LIN {X 0,Y 245.794,Z 1176.659,A -85,B 0,C 180,E1 11030.463,E2 11030.463} C_VEL
LIN {X 0,Y 253.658,Z 1155.772,A -85,B 0,C 180,E1 11026.264,E2 11026.264} C_VEL
LIN {X 0,Y 262.655,Z 1132.428,A -85,B 0,C 180,E1 11022.399,E2 11022.399} C_VEL
LIN {X 0,Y 271.964,Z 1108.253,A -85,B 0,C 180,E1 11019.132,E2 11019.132} C_VEL
LIN {X 0,Y 282.858,Z 1079.724,A -85,B 0,C 180,E1 11015.958,E2 11015.958} C_VEL
LIN {X 0,Y 293.467,Z 1051.429,A -85,B 0,C 180,E1 11013.416,E2 11013.416} C_VEL
LIN {X 0,Y 303.782,Z 1022.552,A -85,B 0,C 180,E1 11011.336,E2 11011.336} C_VEL
LIN {X 0,Y 309.269,Z 1005.972,A -85,B 0,C 180,E1 11010.325,E2 11010.325} C_VEL
LIN {X 0,Y 306.49,Z 980.098,A -85,B 0,C 180,E1 11007.282,E2 11007.282} C_VEL
LIN {X 0,Y 305.142,Z 955.248,A -85,B 0,C 180,E1 11004.695,E2 11004.695} C_VEL
LIN {X 0,Y 304.735,Z 928.08,A -85,B 0,C 180,E1 11002.235,E2 11002.235} C_VEL
LIN {X 0,Y 305.285,Z 899.503,A -85,B 0,C 180,E1 11000.074,E2 11000.074} C_VEL
LIN {X 0,Y 306.681,Z 870.662,A -85,B 0,C 180,E1 10998.043,E2 10998.043} C_VEL
LIN {X 0,Y 314.524,Z 847.538,A -85,B 0,C 180,E1 10995.016,E2 10995.016} C_VEL
LIN {X 0,Y 309.833,Z 833.339,A -85,B 0,C 180,E1 10991.165,E2 10991.165} C_VEL
LIN {X 0,Y 304.885,Z 819.165,A -85,B 0,C 180,E1 10986.97,E2 10986.97} C_VEL
LIN {X 0,Y 300.201,Z 806.583,A -85,B 0,C 180,E1 10982.864,E2 10982.864} C_VEL
LIN {X 0,Y 295.689,Z 794.743,A -85,B 0,C 180,E1 10978.644,E2 10978.644} C_VEL
LIN {X 0,Y 291.025,Z 783.188,A -85,B 0,C 180,E1 10974.084,E2 10974.084} C_VEL
LIN {X 0,Y 286.711,Z 772.817,A -85,B 0,C 180,E1 10969.545,E2 10969.545} C_VEL
LIN {X 0,Y 282.704,Z 763.649,A -85,B 0,C 180,E1 10965.037,E2 10965.037} C_VEL
LIN {X 0,Y 279.359,Z 756.044,A -85,B 0,C 180,E1 10960.884,E2 10960.884} C_VEL
LIN {X 0,Y 276.382,Z 749.179,A -85,B 0,C 180,E1 10956.759,E2 10956.759} C_VEL
LIN {X 0,Y 274.386,Z 744.79,A -85,B 0,C 180,E1 10953.778,E2 10953.778} C_VEL
LIN {X 0,Y 281.502,Z 746.329,A -85,B 0,C 180,E1 10950.823,E2 10950.823} C_VEL
LIN {X 0,Y 285.736,Z 758.772,A -85,B 0,C 180,E1 10947.391,E2 10947.391} C_VEL
LIN {X 0,Y 289.434,Z 771.953,A -85,B 0,C 180,E1 10944.27,E2 10944.27} C_VEL
LIN {X 0,Y 291.796,Z 781.823,A -85,B 0,C 180,E1 10942.234,E2 10942.234} C_VEL
LIN {X 0,Y 283.399,Z 830.233,A -85,B 0,C 180,E1 10937.505,E2 10937.505} C_VEL
LIN {X 0,Y 275.294,Z 882,A -85,B 0,C 180,E1 10932.497,E2 10932.497} C_VEL
LIN {X 0,Y 275.45,Z 888.928,A -85,B 0,C 180,E1 10932.221,E2 10932.221} C_VEL
LIN {X 0,Y 266.995,Z 1035.963,A -85,B 0,C 180,E1 10928.695,E2 10928.695} C_VEL
LIN {X 0,Y 266,Z 1058.102,A -85,B 0,C 180,E1 10927.978,E2 10927.978} C_VEL
LIN {X 0,Y 264.246,Z 1076.059,A -85,B 0,C 180,E1 10927.021,E2 10927.021} C_VEL
LIN {X 0,Y 261.729,Z 1092.625,A -85,B 0,C 180,E1 10925.764,E2 10925.764} C_VEL
LIN {X 0,Y 258.407,Z 1108.653,A -85,B 0,C 180,E1 10924.126,E2 10924.126} C_VEL
LIN {X 0,Y 254.379,Z 1124.313,A -85,B 0,C 180,E1 10922.045,E2 10922.045} C_VEL
LIN {X 0,Y 250.173,Z 1138.097,A -85,B 0,C 180,E1 10919.705,E2 10919.705} C_VEL
LIN {X 0,Y 245.84,Z 1150.471,A -85,B 0,C 180,E1 10917.035,E2 10917.035} C_VEL
LIN {X 0,Y 241.448,Z 1161.815,A -85,B 0,C 180,E1 10913.94,E2 10913.94} C_VEL
LIN {X 0,Y 237.312,Z 1171.782,A -85,B 0,C 180,E1 10910.466,E2 10910.466} C_VEL
LIN {X 0,Y 233.669,Z 1180.12,A -85,B 0,C 180,E1 10906.657,E2 10906.657} C_VEL
LIN {X 0,Y 230.699,Z 1186.833,A -85,B 0,C 180,E1 10902.512,E2 10902.512} C_VEL
LIN {X 0,Y 228.64,Z 1191.633,A -85,B 0,C 180,E1 10898.294,E2 10898.294} C_VEL
LIN {X 0,Y 227.421,Z 1194.668,A -85,B 0,C 180,E1 10894.03,E2 10894.03} C_VEL
LIN {X 0,Y 226.961,Z 1196.042,A -85,B 0,C 180,E1 10889.492,E2 10889.492} C_VEL
LIN {X 0,Y 227.297,Z 1195.648,A -85,B 0,C 180,E1 10884.949,E2 10884.949} C_VEL
LIN {X 0,Y 228.487,Z 1193.456,A -85,B 0,C 180,E1 10880.424,E2 10880.424} C_VEL
LIN {X 0,Y 230.473,Z 1189.568,A -85,B 0,C 180,E1 10876.192,E2 10876.192} C_VEL
LIN {X 0,Y 233.392,Z 1183.816,A -85,B 0,C 180,E1 10872.006,E2 10872.006} C_VEL
LIN {X 0,Y 237.05,Z 1176.45,A -85,B 0,C 180,E1 10868.122,E2 10868.122} C_VEL
LIN {X 0,Y 241.081,Z 1167.875,A -85,B 0,C 180,E1 10864.707,E2 10864.707} C_VEL
LIN {X 0,Y 245.543,Z 1157.661,A -85,B 0,C 180,E1 10861.544,E2 10861.544} C_VEL
LIN {X 0,Y 250.186,Z 1145.999,A -85,B 0,C 180,E1 10858.694,E2 10858.694} C_VEL
LIN {X 0,Y 254.869,Z 1132.781,A -85,B 0,C 180,E1 10856.142,E2 10856.142} C_VEL
LIN {X 0,Y 259.222,Z 1118.358,A -85,B 0,C 180,E1 10853.965,E2 10853.965} C_VEL
LIN {X 0,Y 263.101,Z 1102.793,A -85,B 0,C 180,E1 10852.135,E2 10852.135} C_VEL
LIN {X 0,Y 266.253,Z 1086.649,A -85,B 0,C 180,E1 10850.68,E2 10850.68} C_VEL
LIN {X 0,Y 267.79,Z 1076.701,A -85,B 0,C 180,E1 10849.969,E2 10849.969} C_VEL
LIN {X 0,Y 270.006,Z 1077.25,A -85,B 0,C 180,E1 10849.601,E2 10849.601} C_VEL
LIN {X 0,Y 273.138,Z 1076.234,A -85,B 0,C 180,E1 10849.334,E2 10849.334} C_VEL
LIN {X 0,Y 277.103,Z 1073.311,A -85,B 0,C 180,E1 10849.22,E2 10849.22} C_VEL
LIN {X 0,Y 279.582,Z 1072.671,A -85,B 0,C 180,E1 10848.992,E2 10848.992} C_VEL
LIN {X 0,Y 272.711,Z 1094.804,A -85,B 0,C 180,E1 10846.636,E2 10846.636} C_VEL
LIN {X 0,Y 265.454,Z 1115.949,A -85,B 0,C 180,E1 10843.874,E2 10843.874} C_VEL
LIN {X 0,Y 257.942,Z 1136.201,A -85,B 0,C 180,E1 10840.635,E2 10840.635} C_VEL
LIN {X 0,Y 251.122,Z 1153.816,A -85,B 0,C 180,E1 10837.214,E2 10837.214} C_VEL
LIN {X 0,Y 244.423,Z 1170.711,A -85,B 0,C 180,E1 10833.242,E2 10833.242} C_VEL
LIN {X 0,Y 238.202,Z 1186.646,A -85,B 0,C 180,E1 10828.675,E2 10828.675} C_VEL
LIN {X 0,Y 233.894,Z 1198.218,A -85,B 0,C 180,E1 10824.67,E2 10824.67} C_VEL
LIN {X 0,Y 231.503,Z 1202.313,A -85,B 0,C 180,E1 10823.15,E2 10823.15} C_VEL
LIN {X 0,Y 222.063,Z 1212.153,A -85,B 0,C 180,E1 10819.027,E2 10819.027} C_VEL
LIN {X 0,Y 220.419,Z 1215.207,A -85,B 0,C 180,E1 10817.547,E2 10817.547} C_VEL
LIN {X 0,Y 218.075,Z 1224.725,A -85,B 0,C 180,E1 10812.176,E2 10812.176} C_VEL
LIN {X 0,Y 216.806,Z 1232.767,A -85,B 0,C 180,E1 10806.621,E2 10806.621} C_VEL
LIN {X 0,Y 216.41,Z 1238.955,A -85,B 0,C 180,E1 10801.324,E2 10801.324} C_VEL
LIN {X 0,Y 216.474,Z 1243.705,A -85,B 0,C 180,E1 10796.027,E2 10796.027} C_VEL
LIN {X 0,Y 217.079,Z 1247.526,A -85,B 0,C 180,E1 10790.455,E2 10790.455} C_VEL
LIN {X 0,Y 218.97,Z 1250.36,A -85,B 0,C 180,E1 10784.099,E2 10784.099} C_VEL
LIN {X 0,Y 223.396,Z 1251.95,A -85,B 0,C 180,E1 10777.083,E2 10777.083} C_VEL
LIN {X 0,Y 231.352,Z 1251.855,A -85,B 0,C 180,E1 10769.911,E2 10769.911} C_VEL
LIN {X 0,Y 243.153,Z 1249.952,A -85,B 0,C 180,E1 10763.103,E2 10763.103} C_VEL
LIN {X 0,Y 258.957,Z 1246.212,A -85,B 0,C 180,E1 10756.887,E2 10756.887} C_VEL
LIN {X 0,Y 264.381,Z 1244.756,A -85,B 0,C 180,E1 10755.163,E2 10755.163} C_VEL
LIN {X 0,Y 246.171,Z 1253.178,A -85,B 0,C 180,E1 10749.322,E2 10749.322} C_VEL
LIN {X 0,Y 232.274,Z 1260.245,A -85,B 0,C 180,E1 10742.558,E2 10742.558} C_VEL
LIN {X 0,Y 223.251,Z 1265.258,A -85,B 0,C 180,E1 10735.469,E2 10735.469} C_VEL
LIN {X 0,Y 218.472,Z 1268.085,A -85,B 0,C 180,E1 10728.668,E2 10728.668} C_VEL
LIN {X 0,Y 216.631,Z 1269.015,A -85,B 0,C 180,E1 10722.262,E2 10722.262} C_VEL
LIN {X 0,Y 216.607,Z 1268.218,A -85,B 0,C 180,E1 10716.364,E2 10716.364} C_VEL
LIN {X 0,Y 217.109,Z 1266.169,A -85,B 0,C 180,E1 10711.587,E2 10711.587} C_VEL
LIN {X 0,Y 217.301,Z 1263.421,A -85,B 0,C 180,E1 10707.63,E2 10707.63} C_VEL
LIN {X 0,Y 217.222,Z 1259.203,A -85,B 0,C 180,E1 10703.396,E2 10703.396} C_VEL
LIN {X 0,Y 217.27,Z 1252.953,A -85,B 0,C 180,E1 10698.59,E2 10698.59} C_VEL
LIN {X 0,Y 217.992,Z 1244.563,A -85,B 0,C 180,E1 10693.466,E2 10693.466} C_VEL
LIN {X 0,Y 219.847,Z 1233.738,A -85,B 0,C 180,E1 10688.107,E2 10688.107} C_VEL
LIN {X 0,Y 223.25,Z 1220.001,A -85,B 0,C 180,E1 10682.532,E2 10682.532} C_VEL
LIN {X 0,Y 227.725,Z 1205.387,A -85,B 0,C 180,E1 10677.615,E2 10677.615} C_VEL
LIN {X 0,Y 234.276,Z 1186.649,A -85,B 0,C 180,E1 10672.392,E2 10672.392} C_VEL
LIN {X 0,Y 242.106,Z 1165.933,A -85,B 0,C 180,E1 10667.669,E2 10667.669} C_VEL
LIN {X 0,Y 250.586,Z 1144.273,A -85,B 0,C 180,E1 10663.618,E2 10663.618} C_VEL
LIN {X 0,Y 259.832,Z 1120.935,A -85,B 0,C 180,E1 10660.028,E2 10660.028} C_VEL
LIN {X 0,Y 271.037,Z 1092.34,A -85,B 0,C 180,E1 10656.47,E2 10656.47} C_VEL
LIN {X 0,Y 282.4,Z 1063.011,A -85,B 0,C 180,E1 10653.528,E2 10653.528} C_VEL
LIN {X 0,Y 292.968,Z 1034.784,A -85,B 0,C 180,E1 10651.25,E2 10651.25} C_VEL
LIN {X 0,Y 302.537,Z 1007.602,A -85,B 0,C 180,E1 10649.502,E2 10649.502} C_VEL
LIN {X 0,Y 300.088,Z 981.059,A -85,B 0,C 180,E1 10646.305,E2 10646.305} C_VEL
LIN {X 0,Y 299.039,Z 955.864,A -85,B 0,C 180,E1 10643.637,E2 10643.637} C_VEL
LIN {X 0,Y 299.042,Z 928.661,A -85,B 0,C 180,E1 10641.121,E2 10641.121} C_VEL
LIN {X 0,Y 299.948,Z 898.691,A -85,B 0,C 180,E1 10638.829,E2 10638.829} C_VEL
LIN {X 0,Y 301.641,Z 868.509,A -85,B 0,C 180,E1 10636.679,E2 10636.679} C_VEL
LIN {X 0,Y 307.857,Z 850.994,A -85,B 0,C 180,E1 10634.387,E2 10634.387} C_VEL
LIN {X 0,Y 303,Z 836.151,A -85,B 0,C 180,E1 10630.265,E2 10630.265} C_VEL
LIN {X 0,Y 297.902,Z 821.422,A -85,B 0,C 180,E1 10625.779,E2 10625.779} C_VEL
LIN {X 0,Y 293.033,Z 808.289,A -85,B 0,C 180,E1 10621.363,E2 10621.363} C_VEL
LIN {X 0,Y 288.537,Z 796.595,A -85,B 0,C 180,E1 10617.02,E2 10617.02} C_VEL
LIN {X 0,Y 284.155,Z 785.659,A -85,B 0,C 180,E1 10612.519,E2 10612.519} C_VEL
LIN {X 0,Y 279.79,Z 775.02,A -85,B 0,C 180,E1 10607.618,E2 10607.618} C_VEL
LIN {X 0,Y 275.831,Z 765.954,A -85,B 0,C 180,E1 10602.925,E2 10602.925} C_VEL
LIN {X 0,Y 272.611,Z 758.595,A -85,B 0,C 180,E1 10598.68,E2 10598.68} C_VEL
LIN {X 0,Y 270.256,Z 753.347,A -85,B 0,C 180,E1 10595.287,E2 10595.287} C_VEL
LIN {X 0,Y 269.775,Z 751.899,A -85,B 0,C 180,E1 10594.301,E2 10594.301} C_VEL
LIN {X 0,Y 277.293,Z 753.26,A -85,B 0,C 180,E1 10591.106,E2 10591.106} C_VEL
LIN {X 0,Y 281.203,Z 765.326,A -85,B 0,C 180,E1 10587.767,E2 10587.767} C_VEL
LIN {X 0,Y 284.748,Z 778.734,A -85,B 0,C 180,E1 10584.592,E2 10584.592} C_VEL
LIN {X 0,Y 286.108,Z 785.803,A -85,B 0,C 180,E1 10583.154,E2 10583.154} C_VEL
LIN {X 0,Y 277.26,Z 835.51,A -85,B 0,C 180,E1 10578.284,E2 10578.284} C_VEL
LIN {X 0,Y 269.532,Z 883.178,A -85,B 0,C 180,E1 10573.64,E2 10573.64} C_VEL
LIN {X 0,Y 269.648,Z 889.812,A -85,B 0,C 180,E1 10573.372,E2 10573.372} C_VEL
LIN {X 0,Y 260.896,Z 1036.324,A -85,B 0,C 180,E1 10569.816,E2 10569.816} C_VEL
LIN {X 0,Y 259.821,Z 1059.023,A -85,B 0,C 180,E1 10569.071,E2 10569.071} C_VEL
LIN {X 0,Y 257.987,Z 1077.015,A -85,B 0,C 180,E1 10568.096,E2 10568.096} C_VEL
LIN {X 0,Y 255.337,Z 1093.738,A -85,B 0,C 180,E1 10566.804,E2 10566.804} C_VEL
LIN {X 0,Y 251.881,Z 1109.729,A -85,B 0,C 180,E1 10565.138,E2 10565.138} C_VEL
LIN {X 0,Y 247.896,Z 1124.657,A -85,B 0,C 180,E1 10563.126,E2 10563.126} C_VEL
LIN {X 0,Y 243.507,Z 1138.558,A -85,B 0,C 180,E1 10560.741,E2 10560.741} C_VEL
LIN {X 0,Y 238.88,Z 1151.282,A -85,B 0,C 180,E1 10557.952,E2 10557.952} C_VEL
LIN {X 0,Y 234.216,Z 1162.823,A -85,B 0,C 180,E1 10554.728,E2 10554.728} C_VEL
LIN {X 0,Y 229.89,Z 1172.782,A -85,B 0,C 180,E1 10551.158,E2 10551.158} C_VEL
LIN {X 0,Y 226.071,Z 1181.107,A -85,B 0,C 180,E1 10547.234,E2 10547.234} C_VEL
LIN {X 0,Y 222.952,Z 1187.812,A -85,B 0,C 180,E1 10542.954,E2 10542.954} C_VEL
LIN {X 0,Y 220.784,Z 1192.605,A -85,B 0,C 180,E1 10538.591,E2 10538.591} C_VEL
LIN {X 0,Y 219.5,Z 1195.629,A -85,B 0,C 180,E1 10534.176,E2 10534.176} C_VEL
LIN {X 0,Y 219.018,Z 1196.997,A -85,B 0,C 180,E1 10529.473,E2 10529.473} C_VEL
LIN {X 0,Y 219.38,Z 1196.596,A -85,B 0,C 180,E1 10524.766,E2 10524.766} C_VEL
LIN {X 0,Y 220.549,Z 1194.562,A -85,B 0,C 180,E1 10520.34,E2 10520.34} C_VEL
LIN {X 0,Y 222.602,Z 1190.789,A -85,B 0,C 180,E1 10515.959,E2 10515.959} C_VEL
LIN {X 0,Y 225.604,Z 1185.164,A -85,B 0,C 180,E1 10511.655,E2 10511.655} C_VEL
LIN {X 0,Y 229.328,Z 1178.024,A -85,B 0,C 180,E1 10507.705,E2 10507.705} C_VEL
LIN {X 0,Y 233.599,Z 1169.435,A -85,B 0,C 180,E1 10504.11,E2 10504.11} C_VEL
LIN {X 0,Y 238.433,Z 1158.873,A -85,B 0,C 180,E1 10500.724,E2 10500.724} C_VEL
LIN {X 0,Y 243.421,Z 1146.868,A -85,B 0,C 180,E1 10497.721,E2 10497.721} C_VEL
LIN {X 0,Y 248.299,Z 1133.631,A -85,B 0,C 180,E1 10495.119,E2 10495.119} C_VEL
LIN {X 0,Y 252.828,Z 1119.174,A -85,B 0,C 180,E1 10492.904,E2 10492.904} C_VEL
LIN {X 0,Y 256.861,Z 1103.573,A -85,B 0,C 180,E1 10491.044,E2 10491.044} C_VEL
LIN {X 0,Y 260.061,Z 1087.795,A -85,B 0,C 180,E1 10489.602,E2 10489.602} C_VEL
LIN {X 0,Y 260.438,Z 1086.527,A -85,B 0,C 180,E1 10489.463,E2 10489.463} C_VEL
LIN {X 0,Y 262.674,Z 1087.016,A -85,B 0,C 180,E1 10489.097,E2 10489.097} C_VEL
LIN {X 0,Y 265.828,Z 1086.116,A -85,B 0,C 180,E1 10488.831,E2 10488.831} C_VEL
LIN {X 0,Y 269.275,Z 1084.016,A -85,B 0,C 180,E1 10488.704,E2 10488.704} C_VEL
LIN {X 0,Y 262.103,Z 1105.434,A -85,B 0,C 180,E1 10486.139,E2 10486.139} C_VEL
LIN {X 0,Y 254.799,Z 1125.376,A -85,B 0,C 180,E1 10483.219,E2 10483.219} C_VEL
LIN {X 0,Y 247.46,Z 1144.296,A -85,B 0,C 180,E1 10479.847,E2 10479.847} C_VEL
LIN {X 0,Y 240.208,Z 1162.297,A -85,B 0,C 180,E1 10475.939,E2 10475.939} C_VEL
LIN {X 0,Y 233.451,Z 1178.958,A -85,B 0,C 180,E1 10471.503,E2 10471.503} C_VEL
LIN {X 0,Y 227.863,Z 1193.209,A -85,B 0,C 180,E1 10466.871,E2 10466.871} C_VEL
LIN {X 0,Y 223.258,Z 1206.039,A -85,B 0,C 180,E1 10461.822,E2 10461.822} C_VEL
LIN {X 0,Y 220.419,Z 1215.207,A -85,B 0,C 180,E1 10457.547,E2 10457.547} C_VEL
LIN {X 0,Y 218.514,Z 1218.61,A -85,B 0,C 180,E1 10455.795,E2 10455.795} C_VEL
LIN {X 0,Y 210.171,Z 1227.002,A -85,B 0,C 180,E1 10450.702,E2 10450.702} C_VEL
LIN {X 0,Y 209.282,Z 1228.968,A -85,B 0,C 180,E1 10449.298,E2 10449.298} C_VEL
LIN {X 0,Y 208.522,Z 1235.969,A -85,B 0,C 180,E1 10443.849,E2 10443.849} C_VEL
LIN {X 0,Y 208.4,Z 1241.265,A -85,B 0,C 180,E1 10438.625,E2 10438.625} C_VEL
LIN {X 0,Y 208.698,Z 1245.697,A -85,B 0,C 180,E1 10433.121,E2 10433.121} C_VEL
LIN {X 0,Y 209.938,Z 1249.34,A -85,B 0,C 180,E1 10426.784,E2 10426.784} C_VEL
LIN {X 0,Y 213.367,Z 1251.971,A -85,B 0,C 180,E1 10419.603,E2 10419.603} C_VEL
LIN {X 0,Y 219.89,Z 1253.052,A -85,B 0,C 180,E1 10412.366,E2 10412.366} C_VEL
LIN {X 0,Y 230.592,Z 1252.417,A -85,B 0,C 180,E1 10405.084,E2 10405.084} C_VEL
LIN {X 0,Y 244.926,Z 1250.091,A -85,B 0,C 180,E1 10398.597,E2 10398.597} C_VEL
LIN {X 0,Y 254.57,Z 1248.073,A -85,B 0,C 180,E1 10395.242,E2 10395.242} C_VEL
LIN {X 0,Y 236.892,Z 1255.487,A -85,B 0,C 180,E1 10389.285,E2 10389.285} C_VEL
LIN {X 0,Y 223.172,Z 1261.674,A -85,B 0,C 180,E1 10382.223,E2 10382.223} C_VEL
LIN {X 0,Y 214.434,Z 1265.831,A -85,B 0,C 180,E1 10374.817,E2 10374.817} C_VEL
LIN {X 0,Y 209.919,Z 1267.904,A -85,B 0,C 180,E1 10367.466,E2 10367.466} C_VEL
LIN {X 0,Y 208.558,Z 1268.033,A -85,B 0,C 180,E1 10360.78,E2 10360.78} C_VEL
LIN {X 0,Y 208.816,Z 1266.61,A -85,B 0,C 180,E1 10355.135,E2 10355.135} C_VEL
LIN {X 0,Y 209.308,Z 1264.246,A -85,B 0,C 180,E1 10350.551,E2 10350.551} C_VEL
LIN {X 0,Y 209.402,Z 1260.934,A -85,B 0,C 180,E1 10346.356,E2 10346.356} C_VEL
LIN {X 0,Y 209.286,Z 1255.952,A -85,B 0,C 180,E1 10341.763,E2 10341.763} C_VEL
LIN {X 0,Y 209.539,Z 1248.576,A -85,B 0,C 180,E1 10336.482,E2 10336.482} C_VEL
LIN {X 0,Y 210.665,Z 1239.344,A -85,B 0,C 180,E1 10331.175,E2 10331.175} C_VEL
LIN {X 0,Y 212.966,Z 1228.21,A -85,B 0,C 180,E1 10325.896,E2 10325.896} C_VEL
LIN {X 0,Y 216.825,Z 1214.255,A -85,B 0,C 180,E1 10320.438,E2 10320.438} C_VEL
LIN {X 0,Y 222.236,Z 1197.992,A -85,B 0,C 180,E1 10315.157,E2 10315.157} C_VEL
LIN {X 0,Y 229.421,Z 1178.65,A -85,B 0,C 180,E1 10310,E2 10310} C_VEL
LIN {X 0,Y 237.764,Z 1157.47,A -85,B 0,C 180,E1 10305.394,E2 10305.394} C_VEL
LIN {X 0,Y 246.744,Z 1135.294,A -85,B 0,C 180,E1 10301.443,E2 10301.443} C_VEL
LIN {X 0,Y 256.286,Z 1111.679,A -85,B 0,C 180,E1 10297.998,E2 10297.998} C_VEL
LIN {X 0,Y 267.475,Z 1083.837,A -85,B 0,C 180,E1 10294.679,E2 10294.679} C_VEL
LIN {X 0,Y 278.315,Z 1056.195,A -85,B 0,C 180,E1 10292.026,E2 10292.026} C_VEL
LIN {X 0,Y 289.207,Z 1027.348,A -85,B 0,C 180,E1 10289.804,E2 10289.804} C_VEL
LIN {X 0,Y 295.75,Z 1008.578,A -85,B 0,C 180,E1 10288.581,E2 10288.581} C_VEL
LIN {X 0,Y 293.786,Z 983.697,A -85,B 0,C 180,E1 10285.502,E2 10285.502} C_VEL
LIN {X 0,Y 293.022,Z 956.798,A -85,B 0,C 180,E1 10282.575,E2 10282.575} C_VEL
LIN {X 0,Y 293.271,Z 930.923,A -85,B 0,C 180,E1 10280.142,E2 10280.142} C_VEL
LIN {X 0,Y 294.492,Z 901.692,A -85,B 0,C 180,E1 10277.831,E2 10277.831} C_VEL
LIN {X 0,Y 296.825,Z 865.995,A -85,B 0,C 180,E1 10275.234,E2 10275.234} C_VEL
LIN {X 0,Y 301.092,Z 854.054,A -85,B 0,C 180,E1 10273.638,E2 10273.638} C_VEL
LIN {X 0,Y 296.348,Z 839.521,A -85,B 0,C 180,E1 10269.516,E2 10269.516} C_VEL
LIN {X 0,Y 291.493,Z 825.354,A -85,B 0,C 180,E1 10265.117,E2 10265.117} C_VEL
LIN {X 0,Y 286.894,Z 812.783,A -85,B 0,C 180,E1 10260.799,E2 10260.799} C_VEL
LIN {X 0,Y 282.638,Z 801.557,A -85,B 0,C 180,E1 10256.552,E2 10256.552} C_VEL
LIN {X 0,Y 278.494,Z 791.046,A -85,B 0,C 180,E1 10252.158,E2 10252.158} C_VEL
LIN {X 0,Y 274.106,Z 780.293,A -85,B 0,C 180,E1 10247.143,E2 10247.143} C_VEL
LIN {X 0,Y 270.378,Z 771.57,A -85,B 0,C 180,E1 10242.563,E2 10242.563} C_VEL
LIN {X 0,Y 267.142,Z 764.078,A -85,B 0,C 180,E1 10238.152,E2 10238.152} C_VEL
LIN {X 0,Y 265.106,Z 759.219,A -85,B 0,C 180,E1 10234.893,E2 10234.893} C_VEL
LIN {X 0,Y 273.142,Z 760.371,A -85,B 0,C 180,E1 10231.344,E2 10231.344} C_VEL
LIN {X 0,Y 276.891,Z 772.716,A -85,B 0,C 180,E1 10227.938,E2 10227.938} C_VEL
LIN {X 0,Y 280.124,Z 785.995,A -85,B 0,C 180,E1 10224.82,E2 10224.82} C_VEL
LIN {X 0,Y 280.581,Z 789.263,A -85,B 0,C 180,E1 10224.161,E2 10224.161} C_VEL
LIN {X 0,Y 271.563,Z 838.444,A -85,B 0,C 180,E1 10219.326,E2 10219.326} C_VEL
LIN {X 0,Y 263.87,Z 884.122,A -85,B 0,C 180,E1 10214.845,E2 10214.845} C_VEL
LIN {X 0,Y 263.952,Z 890.793,A -85,B 0,C 180,E1 10214.57,E2 10214.57} C_VEL
LIN {X 0,Y 254.902,Z 1036.681,A -85,B 0,C 180,E1 10210.991,E2 10210.991} C_VEL
LIN {X 0,Y 253.754,Z 1059.803,A -85,B 0,C 180,E1 10210.222,E2 10210.222} C_VEL
LIN {X 0,Y 251.84,Z 1077.842,A -85,B 0,C 180,E1 10209.232,E2 10209.232} C_VEL
LIN {X 0,Y 249.255,Z 1093.661,A -85,B 0,C 180,E1 10208.003,E2 10208.003} C_VEL
LIN {X 0,Y 245.889,Z 1109.065,A -85,B 0,C 180,E1 10206.415,E2 10206.415} C_VEL
LIN {X 0,Y 241.722,Z 1124.29,A -85,B 0,C 180,E1 10204.372,E2 10204.372} C_VEL
LIN {X 0,Y 237.125,Z 1138.418,A -85,B 0,C 180,E1 10201.947,E2 10201.947} C_VEL
LIN {X 0,Y 232.645,Z 1150.457,A -85,B 0,C 180,E1 10199.334,E2 10199.334} C_VEL
LIN {X 0,Y 228.028,Z 1161.596,A -85,B 0,C 180,E1 10196.284,E2 10196.284} C_VEL
LIN {X 0,Y 223.636,Z 1171.327,A -85,B 0,C 180,E1 10192.887,E2 10192.887} C_VEL
LIN {X 0,Y 219.416,Z 1180.198,A -85,B 0,C 180,E1 10188.874,E2 10188.874} C_VEL
LIN {X 0,Y 216.063,Z 1187.102,A -85,B 0,C 180,E1 10184.713,E2 10184.713} C_VEL
LIN {X 0,Y 213.508,Z 1192.357,A -85,B 0,C 180,E1 10180.247,E2 10180.247} C_VEL
LIN {X 0,Y 211.815,Z 1196.005,A -85,B 0,C 180,E1 10175.414,E2 10175.414} C_VEL
LIN {X 0,Y 211.114,Z 1197.824,A -85,B 0,C 180,E1 10170.539,E2 10170.539} C_VEL
LIN {X 0,Y 211.267,Z 1197.863,A -85,B 0,C 180,E1 10165.925,E2 10165.925} C_VEL
LIN {X 0,Y 212.332,Z 1196.109,A -85,B 0,C 180,E1 10161.056,E2 10161.056} C_VEL
LIN {X 0,Y 214.432,Z 1192.508,A -85,B 0,C 180,E1 10156.239,E2 10156.239} C_VEL
LIN {X 0,Y 217.43,Z 1187.254,A -85,B 0,C 180,E1 10151.774,E2 10151.774} C_VEL
LIN {X 0,Y 221.177,Z 1180.425,A -85,B 0,C 180,E1 10147.679,E2 10147.679} C_VEL
LIN {X 0,Y 225.816,Z 1171.569,A -85,B 0,C 180,E1 10143.715,E2 10143.715} C_VEL
LIN {X 0,Y 230.575,Z 1161.836,A -85,B 0,C 180,E1 10140.369,E2 10140.369} C_VEL
LIN {X 0,Y 235.524,Z 1150.69,A -85,B 0,C 180,E1 10137.37,E2 10137.37} C_VEL
LIN {X 0,Y 240.504,Z 1138.028,A -85,B 0,C 180,E1 10134.694,E2 10134.694} C_VEL
LIN {X 0,Y 245.383,Z 1123.73,A -85,B 0,C 180,E1 10132.319,E2 10132.319} C_VEL
LIN {X 0,Y 249.548,Z 1109.16,A -85,B 0,C 180,E1 10130.422,E2 10130.422} C_VEL
LIN {X 0,Y 252.736,Z 1095.469,A -85,B 0,C 180,E1 10129.02,E2 10129.02} C_VEL
LIN {X 0,Y 255.43,Z 1096.005,A -85,B 0,C 180,E1 10128.578,E2 10128.578} C_VEL
LIN {X 0,Y 258.661,Z 1095.233,A -85,B 0,C 180,E1 10128.292,E2 10128.292} C_VEL
LIN {X 0,Y 251.122,Z 1116.176,A -85,B 0,C 180,E1 10125.457,E2 10125.457} C_VEL
LIN {X 0,Y 243.688,Z 1135.319,A -85,B 0,C 180,E1 10122.293,E2 10122.293} C_VEL
LIN {X 0,Y 236.074,Z 1154.036,A -85,B 0,C 180,E1 10118.508,E2 10118.508} C_VEL
LIN {X 0,Y 228.972,Z 1171.068,A -85,B 0,C 180,E1 10114.286,E2 10114.286} C_VEL
LIN {X 0,Y 222.938,Z 1185.758,A -85,B 0,C 180,E1 10109.857,E2 10109.857} C_VEL
LIN {X 0,Y 217.517,Z 1199.775,A -85,B 0,C 180,E1 10104.728,E2 10104.728} C_VEL
LIN {X 0,Y 213.288,Z 1212.232,A -85,B 0,C 180,E1 10099.157,E2 10099.157} C_VEL
LIN {X 0,Y 210.593,Z 1222.215,A -85,B 0,C 180,E1 10093.733,E2 10093.733} C_VEL
LIN {X 0,Y 209.282,Z 1228.968,A -85,B 0,C 180,E1 10089.298,E2 10089.298} C_VEL
LIN {X 0,Y 207.909,Z 1231.679,A -85,B 0,C 180,E1 10087.331,E2 10087.331} C_VEL
LIN {X 0,Y 200.876,Z 1238.211,A -85,B 0,C 180,E1 10081.47,E2 10081.47} C_VEL
LIN {X 0,Y 200.405,Z 1239.563,A -85,B 0,C 180,E1 10080.092,E2 10080.092} C_VEL
LIN {X 0,Y 200.591,Z 1244.571,A -85,B 0,C 180,E1 10074.278,E2 10074.278} C_VEL
LIN {X 0,Y 201.446,Z 1248.313,A -85,B 0,C 180,E1 10068.548,E2 10068.548} C_VEL
LIN {X 0,Y 204.304,Z 1251.692,A -85,B 0,C 180,E1 10061.155,E2 10061.155} C_VEL
LIN {X 0,Y 210.381,Z 1253.636,A -85,B 0,C 180,E1 10053.464,E2 10053.464} C_VEL
LIN {X 0,Y 220.668,Z 1253.909,A -85,B 0,C 180,E1 10045.815,E2 10045.815} C_VEL
LIN {X 0,Y 235.253,Z 1252.428,A -85,B 0,C 180,E1 10038.792,E2 10038.792} C_VEL
LIN {X 0,Y 244.716,Z 1250.961,A -85,B 0,C 180,E1 10035.316,E2 10035.316} C_VEL
LIN {X 0,Y 227.099,Z 1257.595,A -85,B 0,C 180,E1 10029.025,E2 10029.025} C_VEL
LIN {X 0,Y 214.075,Z 1262.738,A -85,B 0,C 180,E1 10021.86,E2 10021.86} C_VEL
LIN {X 0,Y 205.652,Z 1266.056,A -85,B 0,C 180,E1 10014.109,E2 10014.109} C_VEL
LIN {X 0,Y 201.557,Z 1267.336,A -85,B 0,C 180,E1 10006.429,E2 10006.429} C_VEL
LIN {X 0,Y 200.603,Z 1266.762,A -85,B 0,C 180,E1 9999.761,E2 9999.761} C_VEL
LIN {X 0,Y 201.016,Z 1264.945,A -85,B 0,C 180,E1 9994.283,E2 9994.283} C_VEL
LIN {X 0,Y 201.478,Z 1262.316,A -85,B 0,C 180,E1 9989.72,E2 9989.72} C_VEL
LIN {X 0,Y 201.501,Z 1258.641,A -85,B 0,C 180,E1 9985.45,E2 9985.45} C_VEL
LIN {X 0,Y 201.389,Z 1253.123,A -85,B 0,C 180,E1 9980.574,E2 9980.574} C_VEL
LIN {X 0,Y 201.773,Z 1245.658,A -85,B 0,C 180,E1 9975.365,E2 9975.365} C_VEL
LIN {X 0,Y 203.273,Z 1235.355,A -85,B 0,C 180,E1 9969.563,E2 9969.563} C_VEL
LIN {X 0,Y 206.214,Z 1222.811,A -85,B 0,C 180,E1 9963.77,E2 9963.77} C_VEL
LIN {X 0,Y 210.669,Z 1208.176,A -85,B 0,C 180,E1 9958.213,E2 9958.213} C_VEL
LIN {X 0,Y 216.786,Z 1191.036,A -85,B 0,C 180,E1 9952.833,E2 9952.833} C_VEL
LIN {X 0,Y 224.829,Z 1170.497,A -85,B 0,C 180,E1 9947.584,E2 9947.584} C_VEL
LIN {X 0,Y 233.864,Z 1148.503,A -85,B 0,C 180,E1 9943.026,E2 9943.026} C_VEL
LIN {X 0,Y 243.242,Z 1125.918,A -85,B 0,C 180,E1 9939.213,E2 9939.213} C_VEL
LIN {X 0,Y 253.731,Z 1100.486,A -85,B 0,C 180,E1 9935.735,E2 9935.735} C_VEL
LIN {X 0,Y 265.205,Z 1072.315,A -85,B 0,C 180,E1 9932.606,E2 9932.606} C_VEL
LIN {X 0,Y 277.343,Z 1041.625,A -85,B 0,C 180,E1 9929.888,E2 9929.888} C_VEL
LIN {X 0,Y 288.344,Z 1012.353,A -85,B 0,C 180,E1 9927.846,E2 9927.846} C_VEL
LIN {X 0,Y 289.067,Z 1010.058,A -85,B 0,C 180,E1 9927.693,E2 9927.693} C_VEL
LIN {X 0,Y 287.46,Z 986.199,A -85,B 0,C 180,E1 9924.671,E2 9924.671} C_VEL
LIN {X 0,Y 287.015,Z 959.454,A -85,B 0,C 180,E1 9921.671,E2 9921.671} C_VEL
LIN {X 0,Y 287.587,Z 932.564,A -85,B 0,C 180,E1 9919.076,E2 9919.076} C_VEL
LIN {X 0,Y 289.039,Z 904.688,A -85,B 0,C 180,E1 9916.815,E2 9916.815} C_VEL
LIN {X 0,Y 291.91,Z 864.053,A -85,B 0,C 180,E1 9913.833,E2 9913.833} C_VEL
LIN {X 0,Y 294.392,Z 857.419,A -85,B 0,C 180,E1 9912.954,E2 9912.954} C_VEL
LIN {X 0,Y 289.912,Z 843.485,A -85,B 0,C 180,E1 9908.929,E2 9908.929} C_VEL
LIN {X 0,Y 285.318,Z 829.881,A -85,B 0,C 180,E1 9904.623,E2 9904.623} C_VEL
LIN {X 0,Y 280.587,Z 816.704,A -85,B 0,C 180,E1 9900,E2 9900} C_VEL
LIN {X 0,Y 276.161,Z 804.982,A -85,B 0,C 180,E1 9895.431,E2 9895.431} C_VEL
LIN {X 0,Y 272.212,Z 794.961,A -85,B 0,C 180,E1 9891.125,E2 9891.125} C_VEL
LIN {X 0,Y 268.433,Z 785.556,A -85,B 0,C 180,E1 9886.647,E2 9886.647} C_VEL
LIN {X 0,Y 264.839,Z 776.955,A -85,B 0,C 180,E1 9882.055,E2 9882.055} C_VEL
LIN {X 0,Y 261.644,Z 769.435,A -85,B 0,C 180,E1 9877.533,E2 9877.533} C_VEL
LIN {X 0,Y 260.567,Z 766.524,A -85,B 0,C 180,E1 9875.516,E2 9875.516} C_VEL
LIN {X 0,Y 267.681,Z 767.395,A -85,B 0,C 180,E1 9872.165,E2 9872.165} C_VEL
LIN {X 0,Y 269.021,Z 767.568,A -85,B 0,C 180,E1 9871.592,E2 9871.592} C_VEL
LIN {X 0,Y 272.373,Z 779.33,A -85,B 0,C 180,E1 9868.334,E2 9868.334} C_VEL
LIN {X 0,Y 275.312,Z 792.376,A -85,B 0,C 180,E1 9865.267,E2 9865.267} C_VEL
LIN {X 0,Y 265.954,Z 841.349,A -85,B 0,C 180,E1 9860.413,E2 9860.413} C_VEL
LIN {X 0,Y 258.323,Z 884.937,A -85,B 0,C 180,E1 9856.109,E2 9856.109} C_VEL
LIN {X 0,Y 258.39,Z 891.572,A -85,B 0,C 180,E1 9855.826,E2 9855.826} C_VEL
LIN {X 0,Y 249.02,Z 1037.039,A -85,B 0,C 180,E1 9852.221,E2 9852.221} C_VEL
LIN {X 0,Y 247.794,Z 1060.582,A -85,B 0,C 180,E1 9851.43,E2 9851.43} C_VEL
LIN {X 0,Y 245.819,Z 1078.505,A -85,B 0,C 180,E1 9850.435,E2 9850.435} C_VEL
LIN {X 0,Y 243.017,Z 1094.993,A -85,B 0,C 180,E1 9849.136,E2 9849.136} C_VEL
LIN {X 0,Y 239.318,Z 1111.009,A -85,B 0,C 180,E1 9847.434,E2 9847.434} C_VEL
LIN {X 0,Y 234.995,Z 1126.055,A -85,B 0,C 180,E1 9845.353,E2 9845.353} C_VEL
LIN {X 0,Y 230.223,Z 1140.045,A -85,B 0,C 180,E1 9842.876,E2 9842.876} C_VEL
LIN {X 0,Y 225.374,Z 1152.422,A -85,B 0,C 180,E1 9840.084,E2 9840.084} C_VEL
LIN {X 0,Y 220.24,Z 1164.095,A -85,B 0,C 180,E1 9836.705,E2 9836.705} C_VEL
LIN {X 0,Y 215.447,Z 1174.167,A -85,B 0,C 180,E1 9832.94,E2 9832.94} C_VEL
LIN {X 0,Y 211.431,Z 1182.181,A -85,B 0,C 180,E1 9829.041,E2 9829.041} C_VEL
LIN {X 0,Y 208.035,Z 1188.752,A -85,B 0,C 180,E1 9824.754,E2 9824.754} C_VEL
LIN {X 0,Y 205.441,Z 1193.817,A -85,B 0,C 180,E1 9820.087,E2 9820.087} C_VEL
LIN {X 0,Y 203.78,Z 1197.278,A -85,B 0,C 180,E1 9815.063,E2 9815.063} C_VEL
LIN {X 0,Y 203.158,Z 1198.836,A -85,B 0,C 180,E1 9810.278,E2 9810.278} C_VEL
LIN {X 0,Y 203.414,Z 1198.683,A -85,B 0,C 180,E1 9805.203,E2 9805.203} C_VEL
LIN {X 0,Y 204.67,Z 1196.748,A -85,B 0,C 180,E1 9800.151,E2 9800.151} C_VEL
LIN {X 0,Y 206.868,Z 1193.199,A -85,B 0,C 180,E1 9795.44,E2 9795.44} C_VEL
LIN {X 0,Y 210.099,Z 1187.787,A -85,B 0,C 180,E1 9790.826,E2 9790.826} C_VEL
LIN {X 0,Y 214.109,Z 1180.842,A -85,B 0,C 180,E1 9786.609,E2 9786.609} C_VEL
LIN {X 0,Y 218.706,Z 1172.471,A -85,B 0,C 180,E1 9782.791,E2 9782.791} C_VEL
LIN {X 0,Y 223.69,Z 1162.727,A -85,B 0,C 180,E1 9779.361,E2 9779.361} C_VEL
LIN {X 0,Y 228.86,Z 1151.56,A -85,B 0,C 180,E1 9776.295,E2 9776.295} C_VEL
LIN {X 0,Y 234.053,Z 1138.88,A -85,B 0,C 180,E1 9773.568,E2 9773.568} C_VEL
LIN {X 0,Y 239.133,Z 1124.559,A -85,B 0,C 180,E1 9771.153,E2 9771.153} C_VEL
LIN {X 0,Y 243.465,Z 1109.958,A -85,B 0,C 180,E1 9769.228,E2 9769.228} C_VEL
LIN {X 0,Y 245.069,Z 1103.867,A -85,B 0,C 180,E1 9768.545,E2 9768.545} C_VEL
LIN {X 0,Y 247.31,Z 1104.403,A -85,B 0,C 180,E1 9768.152,E2 9768.152} C_VEL
LIN {X 0,Y 248.413,Z 1104.49,A -85,B 0,C 180,E1 9767.994,E2 9767.994} C_VEL
LIN {X 0,Y 240.389,Z 1125.421,A -85,B 0,C 180,E1 9764.832,E2 9764.832} C_VEL
LIN {X 0,Y 232.257,Z 1145.341,A -85,B 0,C 180,E1 9761.111,E2 9761.111} C_VEL
LIN {X 0,Y 224.594,Z 1163.368,A -85,B 0,C 180,E1 9756.943,E2 9756.943} C_VEL
LIN {X 0,Y 217.871,Z 1179.145,A -85,B 0,C 180,E1 9752.477,E2 9752.477} C_VEL
LIN {X 0,Y 211.965,Z 1193.572,A -85,B 0,C 180,E1 9747.515,E2 9747.515} C_VEL
LIN {X 0,Y 206.97,Z 1207.035,A -85,B 0,C 180,E1 9741.839,E2 9741.839} C_VEL
LIN {X 0,Y 203.487,Z 1218.394,A -85,B 0,C 180,E1 9735.972,E2 9735.972} C_VEL
LIN {X 0,Y 201.505,Z 1227.421,A -85,B 0,C 180,E1 9730.29,E2 9730.29} C_VEL
LIN {X 0,Y 200.581,Z 1234.775,A -85,B 0,C 180,E1 9724.575,E2 9724.575} C_VEL
LIN {X 0,Y 200.405,Z 1239.563,A -85,B 0,C 180,E1 9720.092,E2 9720.092} C_VEL
LIN {X 0,Y 199.535,Z 1241.421,A -85,B 0,C 180,E1 9718.115,E2 9718.115} C_VEL
LIN {X 0,Y 196.024,Z 1244.022,A -85,B 0,C 180,E1 9714.779,E2 9714.779} C_VEL
LIN {X 0,Y 193.274,Z 1246.233,A -85,B 0,C 180,E1 9711.454,E2 9711.454} C_VEL
LIN {X 0,Y 193.109,Z 1247.098,A -85,B 0,C 180,E1 9710.148,E2 9710.148} C_VEL
LIN {X 0,Y 195.408,Z 1251.042,A -85,B 0,C 180,E1 9702.735,E2 9702.735} C_VEL
LIN {X 0,Y 201.19,Z 1253.872,A -85,B 0,C 180,E1 9694.381,E2 9694.381} C_VEL
LIN {X 0,Y 211.551,Z 1254.985,A -85,B 0,C 180,E1 9686.101,E2 9686.101} C_VEL
LIN {X 0,Y 226.619,Z 1254.281,A -85,B 0,C 180,E1 9678.56,E2 9678.56} C_VEL
LIN {X 0,Y 234.878,Z 1253.409,A -85,B 0,C 180,E1 9675.407,E2 9675.407} C_VEL
LIN {X 0,Y 217.316,Z 1259.268,A -85,B 0,C 180,E1 9668.741,E2 9668.741} C_VEL
LIN {X 0,Y 204.638,Z 1263.54,A -85,B 0,C 180,E1 9661.198,E2 9661.198} C_VEL
LIN {X 0,Y 196.719,Z 1265.973,A -85,B 0,C 180,E1 9653.044,E2 9653.044} C_VEL
LIN {X 0,Y 193.219,Z 1266.401,A -85,B 0,C 180,E1 9645,E2 9645} C_VEL
LIN {X 0,Y 192.743,Z 1265.151,A -85,B 0,C 180,E1 9638.356,E2 9638.356} C_VEL
LIN {X 0,Y 193.295,Z 1262.896,A -85,B 0,C 180,E1 9632.969,E2 9632.969} C_VEL
LIN {X 0,Y 193.645,Z 1260.144,A -85,B 0,C 180,E1 9628.821,E2 9628.821} C_VEL
LIN {X 0,Y 193.575,Z 1256.119,A -85,B 0,C 180,E1 9624.372,E2 9624.372} C_VEL
LIN {X 0,Y 193.53,Z 1249.701,A -85,B 0,C 180,E1 9618.984,E2 9618.984} C_VEL
LIN {X 0,Y 194.249,Z 1241.027,A -85,B 0,C 180,E1 9613.222,E2 9613.222} C_VEL
LIN {X 0,Y 196.141,Z 1230.53,A -85,B 0,C 180,E1 9607.526,E2 9607.526} C_VEL
LIN {X 0,Y 199.65,Z 1217.303,A -85,B 0,C 180,E1 9601.595,E2 9601.595} C_VEL
LIN {X 0,Y 204.529,Z 1202.571,A -85,B 0,C 180,E1 9596.135,E2 9596.135} C_VEL
LIN {X 0,Y 211.708,Z 1183.673,A -85,B 0,C 180,E1 9590.392,E2 9590.392} C_VEL
LIN {X 0,Y 220.02,Z 1163.408,A -85,B 0,C 180,E1 9585.408,E2 9585.408} C_VEL
LIN {X 0,Y 229.292,Z 1141.524,A -85,B 0,C 180,E1 9581.032,E2 9581.032} C_VEL
LIN {X 0,Y 239.548,Z 1117.444,A -85,B 0,C 180,E1 9577.138,E2 9577.138} C_VEL
LIN {X 0,Y 251.939,Z 1087.916,A -85,B 0,C 180,E1 9573.346,E2 9573.346} C_VEL
LIN {X 0,Y 264.469,Z 1057.542,A -85,B 0,C 180,E1 9570.25,E2 9570.25} C_VEL
LIN {X 0,Y 275.661,Z 1029.406,A -85,B 0,C 180,E1 9567.973,E2 9567.973} C_VEL
LIN {X 0,Y 282.355,Z 1011.136,A -85,B 0,C 180,E1 9566.727,E2 9566.727} C_VEL
LIN {X 0,Y 281.046,Z 985.922,A -85,B 0,C 180,E1 9563.483,E2 9563.483} C_VEL
LIN {X 0,Y 281.052,Z 959.912,A -85,B 0,C 180,E1 9560.514,E2 9560.514} C_VEL
LIN {X 0,Y 282.039,Z 931.594,A -85,B 0,C 180,E1 9557.752,E2 9557.752} C_VEL
LIN {X 0,Y 283.848,Z 904.149,A -85,B 0,C 180,E1 9555.502,E2 9555.502} C_VEL
LIN {X 0,Y 287.183,Z 861.849,A -85,B 0,C 180,E1 9552.364,E2 9552.364} C_VEL
LIN {X 0,Y 287.625,Z 860.382,A -85,B 0,C 180,E1 9552.141,E2 9552.141} C_VEL
LIN {X 0,Y 282.889,Z 845.561,A -85,B 0,C 180,E1 9547.719,E2 9547.719} C_VEL
LIN {X 0,Y 278.333,Z 832.037,A -85,B 0,C 180,E1 9543.295,E2 9543.295} C_VEL
LIN {X 0,Y 273.625,Z 818.901,A -85,B 0,C 180,E1 9538.534,E2 9538.534} C_VEL
LIN {X 0,Y 269.419,Z 807.732,A -85,B 0,C 180,E1 9534.019,E2 9534.019} C_VEL
LIN {X 0,Y 265.588,Z 797.834,A -85,B 0,C 180,E1 9529.589,E2 9529.589} C_VEL
LIN {X 0,Y 261.755,Z 788.09,A -85,B 0,C 180,E1 9524.717,E2 9524.717} C_VEL
LIN {X 0,Y 258.15,Z 779.494,A -85,B 0,C 180,E1 9519.835,E2 9519.835} C_VEL
LIN {X 0,Y 255.844,Z 773.796,A -85,B 0,C 180,E1 9516.262,E2 9516.262} C_VEL
LIN {X 0,Y 264.159,Z 774.687,A -85,B 0,C 180,E1 9512.252,E2 9512.252} C_VEL
LIN {X 0,Y 265.036,Z 774.833,A -85,B 0,C 180,E1 9511.863,E2 9511.863} C_VEL
LIN {X 0,Y 268.082,Z 786.435,A -85,B 0,C 180,E1 9508.656,E2 9508.656} C_VEL
LIN {X 0,Y 270,Z 796.275,A -85,B 0,C 180,E1 9506.331,E2 9506.331} C_VEL
LIN {X 0,Y 260.232,Z 845.464,A -85,B 0,C 180,E1 9501.43,E2 9501.43} C_VEL
LIN {X 0,Y 252.919,Z 886.037,A -85,B 0,C 180,E1 9497.412,E2 9497.412} C_VEL
LIN {X 0,Y 252.943,Z 892.562,A -85,B 0,C 180,E1 9497.131,E2 9497.131} C_VEL
LIN {X 0,Y 243.258,Z 1037.397,A -85,B 0,C 180,E1 9493.511,E2 9493.511} C_VEL
LIN {X 0,Y 241.946,Z 1061.406,A -85,B 0,C 180,E1 9492.694,E2 9492.694} C_VEL
LIN {X 0,Y 239.896,Z 1079.273,A -85,B 0,C 180,E1 9491.692,E2 9491.692} C_VEL
LIN {X 0,Y 236.897,Z 1096.227,A -85,B 0,C 180,E1 9490.336,E2 9490.336} C_VEL
LIN {X 0,Y 233.07,Z 1112.084,A -85,B 0,C 180,E1 9488.619,E2 9488.619} C_VEL
LIN {X 0,Y 228.572,Z 1127.109,A -85,B 0,C 180,E1 9486.503,E2 9486.503} C_VEL
LIN {X 0,Y 223.602,Z 1141.083,A -85,B 0,C 180,E1 9483.98,E2 9483.98} C_VEL
LIN {X 0,Y 218.544,Z 1153.441,A -85,B 0,C 180,E1 9481.127,E2 9481.127} C_VEL
LIN {X 0,Y 213.179,Z 1165.103,A -85,B 0,C 180,E1 9477.663,E2 9477.663} C_VEL
LIN {X 0,Y 208.159,Z 1175.166,A -85,B 0,C 180,E1 9473.792,E2 9473.792} C_VEL
LIN {X 0,Y 203.77,Z 1183.479,A -85,B 0,C 180,E1 9469.586,E2 9469.586} C_VEL
LIN {X 0,Y 200.172,Z 1190.071,A -85,B 0,C 180,E1 9465.051,E2 9465.051} C_VEL
LIN {X 0,Y 197.499,Z 1195.033,A -85,B 0,C 180,E1 9460.202,E2 9460.202} C_VEL
LIN {X 0,Y 195.871,Z 1198.242,A -85,B 0,C 180,E1 9455.268,E2 9455.268} C_VEL
LIN {X 0,Y 195.215,Z 1199.791,A -85,B 0,C 180,E1 9450.289,E2 9450.289} C_VEL
LIN {X 0,Y 195.494,Z 1199.631,A -85,B 0,C 180,E1 9445.008,E2 9445.008} C_VEL
LIN {X 0,Y 196.837,Z 1197.689,A -85,B 0,C 180,E1 9439.755,E2 9439.755} C_VEL
LIN {X 0,Y 199.173,Z 1194.134,A -85,B 0,C 180,E1 9434.864,E2 9434.864} C_VEL
LIN {X 0,Y 202.594,Z 1188.71,A -85,B 0,C 180,E1 9430.086,E2 9430.086} C_VEL
LIN {X 0,Y 206.824,Z 1181.756,A -85,B 0,C 180,E1 9425.733,E2 9425.733} C_VEL
LIN {X 0,Y 211.656,Z 1173.375,A -85,B 0,C 180,E1 9421.805,E2 9421.805} C_VEL
LIN {X 0,Y 216.878,Z 1163.618,A -85,B 0,C 180,E1 9418.289,E2 9418.289} C_VEL
LIN {X 0,Y 222.281,Z 1152.43,A -85,B 0,C 180,E1 9415.156,E2 9415.156} C_VEL
LIN {X 0,Y 227.699,Z 1139.733,A -85,B 0,C 180,E1 9412.379,E2 9412.379} C_VEL
LIN {X 0,Y 232.988,Z 1125.389,A -85,B 0,C 180,E1 9409.925,E2 9409.925} C_VEL
LIN {X 0,Y 237.404,Z 1111.632,A -85,B 0,C 180,E1 9408.036,E2 9408.036} C_VEL
LIN {X 0,Y 238.443,Z 1112.214,A -85,B 0,C 180,E1 9407.788,E2 9407.788} C_VEL
LIN {X 0,Y 230.438,Z 1132.059,A -85,B 0,C 180,E1 9404.488,E2 9404.488} C_VEL
LIN {X 0,Y 222.479,Z 1150.76,A -85,B 0,C 180,E1 9400.668,E2 9400.668} C_VEL
LIN {X 0,Y 215.192,Z 1167.457,A -85,B 0,C 180,E1 9396.495,E2 9396.495} C_VEL
LIN {X 0,Y 208.561,Z 1182.793,A -85,B 0,C 180,E1 9391.828,E2 9391.828} C_VEL
LIN {X 0,Y 202.562,Z 1197.412,A -85,B 0,C 180,E1 9386.376,E2 9386.376} C_VEL
LIN {X 0,Y 198.042,Z 1209.774,A -85,B 0,C 180,E1 9380.697,E2 9380.697} C_VEL
LIN {X 0,Y 194.844,Z 1220.719,A -85,B 0,C 180,E1 9374.564,E2 9374.564} C_VEL
LIN {X 0,Y 193.078,Z 1229.796,A -85,B 0,C 180,E1 9368.338,E2 9368.338} C_VEL
LIN {X 0,Y 192.468,Z 1236.523,A -85,B 0,C 180,E1 9362.68,E2 9362.68} C_VEL
LIN {X 0,Y 192.443,Z 1241.979,A -85,B 0,C 180,E1 9357.022,E2 9357.022} C_VEL
LIN {X 0,Y 192.964,Z 1246.484,A -85,B 0,C 180,E1 9351.057,E2 9351.057} C_VEL
LIN {X 0,Y 193.109,Z 1247.098,A -85,B 0,C 180,E1 9350.148,E2 9350.148} C_VEL
LIN {X 0,Y 192.558,Z 1248.496,A -85,B 0,C 180,E1 9347.885,E2 9347.885} C_VEL
LIN {X 0,Y 188.556,Z 1251.523,A -85,B 0,C 180,E1 9341.314,E2 9341.314} C_VEL
LIN {X 0,Y 188.962,Z 1252.219,A -85,B 0,C 180,E1 9339.639,E2 9339.639} C_VEL
LIN {X 0,Y 196.304,Z 1254.941,A -85,B 0,C 180,E1 9331.06,E2 9331.06} C_VEL
LIN {X 0,Y 208.612,Z 1256.025,A -85,B 0,C 180,E1 9322.722,E2 9322.722} C_VEL
LIN {X 0,Y 225.034,Z 1255.435,A -85,B 0,C 180,E1 9315.496,E2 9315.496} C_VEL
LIN {X 0,Y 207.55,Z 1260.517,A -85,B 0,C 180,E1 9308.428,E2 9308.428} C_VEL
LIN {X 0,Y 195.256,Z 1263.927,A -85,B 0,C 180,E1 9300.466,E2 9300.466} C_VEL
LIN {X 0,Y 187.889,Z 1265.487,A -85,B 0,C 180,E1 9291.875,E2 9291.875} C_VEL
LIN {X 0,Y 185.063,Z 1265.118,A -85,B 0,C 180,E1 9283.757,E2 9283.757} C_VEL
LIN {X 0,Y 184.99,Z 1263.221,A -85,B 0,C 180,E1 9276.833,E2 9276.833} C_VEL
LIN {X 0,Y 185.602,Z 1260.57,A -85,B 0,C 180,E1 9271.548,E2 9271.548} C_VEL
LIN {X 0,Y 185.796,Z 1257.282,A -85,B 0,C 180,E1 9267.228,E2 9267.228} C_VEL
LIN {X 0,Y 185.624,Z 1252.306,A -85,B 0,C 180,E1 9262.265,E2 9262.265} C_VEL
LIN {X 0,Y 185.802,Z 1245.061,A -85,B 0,C 180,E1 9256.625,E2 9256.625} C_VEL
LIN {X 0,Y 186.995,Z 1235.545,A -85,B 0,C 180,E1 9250.643,E2 9250.643} C_VEL
LIN {X 0,Y 189.733,Z 1223.408,A -85,B 0,C 180,E1 9244.402,E2 9244.402} C_VEL
LIN {X 0,Y 194.167,Z 1209.035,A -85,B 0,C 180,E1 9238.319,E2 9238.319} C_VEL
LIN {X 0,Y 200.366,Z 1192.197,A -85,B 0,C 180,E1 9232.501,E2 9232.501} C_VEL
LIN {X 0,Y 207.89,Z 1173.825,A -85,B 0,C 180,E1 9227.305,E2 9227.305} C_VEL
LIN {X 0,Y 217.414,Z 1151.671,A -85,B 0,C 180,E1 9222.237,E2 9222.237} C_VEL
LIN {X 0,Y 228.205,Z 1126.974,A -85,B 0,C 180,E1 9217.74,E2 9217.74} C_VEL
LIN {X 0,Y 239.282,Z 1101.354,A -85,B 0,C 180,E1 9214.052,E2 9214.052} C_VEL
LIN {X 0,Y 252.05,Z 1071.402,A -85,B 0,C 180,E1 9210.596,E2 9210.596} C_VEL
LIN {X 0,Y 264.207,Z 1042.038,A -85,B 0,C 180,E1 9207.919,E2 9207.919} C_VEL
LIN {X 0,Y 275.728,Z 1012.665,A -85,B 0,C 180,E1 9205.796,E2 9205.796} C_VEL
LIN {X 0,Y 274.74,Z 986.454,A -85,B 0,C 180,E1 9202.354,E2 9202.354} C_VEL
LIN {X 0,Y 275.159,Z 959.155,A -85,B 0,C 180,E1 9199.2,E2 9199.2} C_VEL
LIN {X 0,Y 276.555,Z 931.159,A -85,B 0,C 180,E1 9196.44,E2 9196.44} C_VEL
LIN {X 0,Y 278.831,Z 902.14,A -85,B 0,C 180,E1 9194.048,E2 9194.048} C_VEL
LIN {X 0,Y 281.943,Z 864.382,A -85,B 0,C 180,E1 9191.196,E2 9191.196} C_VEL
LIN {X 0,Y 279.162,Z 857.93,A -85,B 0,C 180,E1 9189.691,E2 9189.691} C_VEL
LIN {X 0,Y 274.41,Z 843.16,A -85,B 0,C 180,E1 9185.017,E2 9185.017} C_VEL
LIN {X 0,Y 269.925,Z 830.092,A -85,B 0,C 180,E1 9180.424,E2 9180.424} C_VEL
LIN {X 0,Y 265.532,Z 817.886,A -85,B 0,C 180,E1 9175.681,E2 9175.681} C_VEL
LIN {X 0,Y 261.647,Z 807.545,A -85,B 0,C 180,E1 9171.207,E2 9171.207} C_VEL
LIN {X 0,Y 257.718,Z 797.397,A -85,B 0,C 180,E1 9166.31,E2 9166.31} C_VEL
LIN {X 0,Y 254.469,Z 789.319,A -85,B 0,C 180,E1 9161.916,E2 9161.916} C_VEL
LIN {X 0,Y 251.388,Z 781.774,A -85,B 0,C 180,E1 9157.305,E2 9157.305} C_VEL
LIN {X 0,Y 251.276,Z 781.31,A -85,B 0,C 180,E1 9156.924,E2 9156.924} C_VEL
LIN {X 0,Y 260.638,Z 781.981,A -85,B 0,C 180,E1 9152.342,E2 9152.342} C_VEL
LIN {X 0,Y 261.058,Z 782.096,A -85,B 0,C 180,E1 9152.142,E2 9152.142} C_VEL
LIN {X 0,Y 263.695,Z 793.613,A -85,B 0,C 180,E1 9148.956,E2 9148.956} C_VEL
LIN {X 0,Y 264.776,Z 799.91,A -85,B 0,C 180,E1 9147.459,E2 9147.459} C_VEL
LIN {X 0,Y 254.859,Z 848.7,A -85,B 0,C 180,E1 9142.599,E2 9142.599} C_VEL
LIN {X 0,Y 247.654,Z 887.218,A -85,B 0,C 180,E1 9138.767,E2 9138.767} C_VEL
LIN {X 0,Y 247.624,Z 893.668,A -85,B 0,C 180,E1 9138.49,E2 9138.49} C_VEL
LIN {X 0,Y 237.625,Z 1037.751,A -85,B 0,C 180,E1 9134.862,E2 9134.862} C_VEL
LIN {X 0,Y 236.221,Z 1062.232,A -85,B 0,C 180,E1 9134.02,E2 9134.02} C_VEL
LIN {X 0,Y 234.096,Z 1080.04,A -85,B 0,C 180,E1 9133.011,E2 9133.011} C_VEL
LIN {X 0,Y 231.224,Z 1095.801,A -85,B 0,C 180,E1 9131.75,E2 9131.75} C_VEL
LIN {X 0,Y 227.474,Z 1111.279,A -85,B 0,C 180,E1 9130.107,E2 9130.107} C_VEL
LIN {X 0,Y 222.976,Z 1126.028,A -85,B 0,C 180,E1 9128.062,E2 9128.062} C_VEL
LIN {X 0,Y 217.756,Z 1140.353,A -85,B 0,C 180,E1 9125.506,E2 9125.506} C_VEL
LIN {X 0,Y 212.215,Z 1153.531,A -85,B 0,C 180,E1 9122.484,E2 9122.484} C_VEL
LIN {X 0,Y 206.946,Z 1164.62,A -85,B 0,C 180,E1 9119.204,E2 9119.204} C_VEL
LIN {X 0,Y 201.572,Z 1174.937,A -85,B 0,C 180,E1 9115.247,E2 9115.247} C_VEL
LIN {X 0,Y 196.753,Z 1183.668,A -85,B 0,C 180,E1 9110.834,E2 9110.834} C_VEL
LIN {X 0,Y 192.923,Z 1190.37,A -85,B 0,C 180,E1 9106.248,E2 9106.248} C_VEL
LIN {X 0,Y 189.962,Z 1195.517,A -85,B 0,C 180,E1 9101.226,E2 9101.226} C_VEL
LIN {X 0,Y 188.035,Z 1199.053,A -85,B 0,C 180,E1 9095.794,E2 9095.794} C_VEL
LIN {X 0,Y 187.271,Z 1200.746,A -85,B 0,C 180,E1 9090.302,E2 9090.302} C_VEL
LIN {X 0,Y 187.576,Z 1200.579,A -85,B 0,C 180,E1 9084.797,E2 9084.797} C_VEL
LIN {X 0,Y 189.014,Z 1198.631,A -85,B 0,C 180,E1 9079.326,E2 9079.326} C_VEL
LIN {X 0,Y 191.5,Z 1195.069,A -85,B 0,C 180,E1 9074.242,E2 9074.242} C_VEL
LIN {X 0,Y 195.125,Z 1189.632,A -85,B 0,C 180,E1 9069.29,E2 9069.29} C_VEL
LIN {X 0,Y 199.905,Z 1182.173,A -85,B 0,C 180,E1 9064.519,E2 9064.519} C_VEL
LIN {X 0,Y 205.045,Z 1173.663,A -85,B 0,C 180,E1 9060.49,E2 9060.49} C_VEL
LIN {X 0,Y 210.564,Z 1163.723,A -85,B 0,C 180,E1 9056.897,E2 9056.897} C_VEL
LIN {X 0,Y 216.249,Z 1152.316,A -85,B 0,C 180,E1 9053.708,E2 9053.708} C_VEL
LIN {X 0,Y 222.183,Z 1138.812,A -85,B 0,C 180,E1 9050.777,E2 9050.777} C_VEL
LIN {X 0,Y 227.472,Z 1124.783,A -85,B 0,C 180,E1 9048.41,E2 9048.41} C_VEL
LIN {X 0,Y 228.874,Z 1120.164,A -85,B 0,C 180,E1 9047.728,E2 9047.728} C_VEL
LIN {X 0,Y 228.22,Z 1120.045,A -85,B 0,C 180,E1 9047.471,E2 9047.471} C_VEL
LIN {X 0,Y 220.219,Z 1138.967,A -85,B 0,C 180,E1 9044.003,E2 9044.003} C_VEL
LIN {X 0,Y 212.12,Z 1157.294,A -85,B 0,C 180,E1 9039.872,E2 9039.872} C_VEL
LIN {X 0,Y 204.614,Z 1174.032,A -85,B 0,C 180,E1 9035.214,E2 9035.214} C_VEL
LIN {X 0,Y 197.971,Z 1189.2,A -85,B 0,C 180,E1 9030.001,E2 9030.001} C_VEL
LIN {X 0,Y 192.696,Z 1202.25,A -85,B 0,C 180,E1 9024.527,E2 9024.527} C_VEL
LIN {X 0,Y 188.472,Z 1214.508,A -85,B 0,C 180,E1 9018.241,E2 9018.241} C_VEL
LIN {X 0,Y 185.965,Z 1224.35,A -85,B 0,C 180,E1 9012.105,E2 9012.105} C_VEL
LIN {X 0,Y 184.73,Z 1232.423,A -85,B 0,C 180,E1 9005.903,E2 9005.903} C_VEL
LIN {X 0,Y 184.428,Z 1239.063,A -85,B 0,C 180,E1 8999.689,E2 8999.689} C_VEL
LIN {X 0,Y 184.648,Z 1244.086,A -85,B 0,C 180,E1 8993.783,E2 8993.783} C_VEL
LIN {X 0,Y 185.822,Z 1248.693,A -85,B 0,C 180,E1 8986.907,E2 8986.907} C_VEL
LIN {X 0,Y 188.962,Z 1252.219,A -85,B 0,C 180,E1 8979.639,E2 8979.639} C_VEL
LIN {X 0,Y 189.505,Z 1253.162,A -85,B 0,C 180,E1 8977.312,E2 8977.312} C_VEL
LIN {X 0,Y 188.929,Z 1255.263,A -85,B 0,C 180,E1 8970.736,E2 8970.736} C_VEL
LIN {X 0,Y 190.351,Z 1255.695,A -85,B 0,C 180,E1 8968.946,E2 8968.946} C_VEL
LIN {X 0,Y 203.545,Z 1257.038,A -85,B 0,C 180,E1 8960.676,E2 8960.676} C_VEL
LIN {X 0,Y 215.243,Z 1257.035,A -85,B 0,C 180,E1 8955.597,E2 8955.597} C_VEL
LIN {X 0,Y 197.804,Z 1261.343,A -85,B 0,C 180,E1 8948.08,E2 8948.08} C_VEL
LIN {X 0,Y 185.61,Z 1263.964,A -85,B 0,C 180,E1 8939.359,E2 8939.359} C_VEL
LIN {X 0,Y 178.981,Z 1264.613,A -85,B 0,C 180,E1 8930.191,E2 8930.191} C_VEL
LIN {X 0,Y 176.987,Z 1263.444,A -85,B 0,C 180,E1 8922.07,E2 8922.07} C_VEL
LIN {X 0,Y 177.318,Z 1260.961,A -85,B 0,C 180,E1 8915.181,E2 8915.181} C_VEL
LIN {X 0,Y 177.886,Z 1258.129,A -85,B 0,C 180,E1 8910.326,E2 8910.326} C_VEL
LIN {X 0,Y 177.908,Z 1254.401,A -85,B 0,C 180,E1 8905.814,E2 8905.814} C_VEL
LIN {X 0,Y 177.739,Z 1248.821,A -85,B 0,C 180,E1 8900.615,E2 8900.615} C_VEL
LIN {X 0,Y 178.157,Z 1240.925,A -85,B 0,C 180,E1 8894.71,E2 8894.71} C_VEL
LIN {X 0,Y 179.933,Z 1230.105,A -85,B 0,C 180,E1 8888.129,E2 8888.129} C_VEL
LIN {X 0,Y 184.968,Z 1212.738,A -85,B 0,C 180,E1 8879.465,E2 8879.465} C_VEL
LIN {X 0,Y 188.975,Z 1201.495,A -85,B 0,C 180,E1 8875.098,E2 8875.098} C_VEL
LIN {X 0,Y 199.712,Z 1174.637,A -85,B 0,C 180,E1 8866.968,E2 8866.968} C_VEL
LIN {X 0,Y 208.952,Z 1153.635,A -85,B 0,C 180,E1 8861.924,E2 8861.924} C_VEL
LIN {X 0,Y 218.68,Z 1131.966,A -85,B 0,C 180,E1 8857.726,E2 8857.726} C_VEL
LIN {X 0,Y 229.877,Z 1106.8,A -85,B 0,C 180,E1 8853.828,E2 8853.828} C_VEL
LIN {X 0,Y 242.878,Z 1077.109,A -85,B 0,C 180,E1 8850.178,E2 8850.178} C_VEL
LIN {X 0,Y 255.857,Z 1046.676,A -85,B 0,C 180,E1 8847.252,E2 8847.252} C_VEL
LIN {X 0,Y 268.046,Z 1016.59,A -85,B 0,C 180,E1 8844.988,E2 8844.988} C_VEL
LIN {X 0,Y 269.086,Z 1013.655,A -85,B 0,C 180,E1 8844.769,E2 8844.769} C_VEL
LIN {X 0,Y 268.501,Z 985.899,A -85,B 0,C 180,E1 8841.061,E2 8841.061} C_VEL
LIN {X 0,Y 269.19,Z 961.377,A -85,B 0,C 180,E1 8838.181,E2 8838.181} C_VEL
LIN {X 0,Y 271.012,Z 933.003,A -85,B 0,C 180,E1 8835.296,E2 8835.296} C_VEL
LIN {X 0,Y 273.492,Z 904.656,A -85,B 0,C 180,E1 8832.913,E2 8832.913} C_VEL
LIN {X 0,Y 276.751,Z 868.519,A -85,B 0,C 180,E1 8830.145,E2 8830.145} C_VEL
LIN {X 0,Y 270.026,Z 853.315,A -85,B 0,C 180,E1 8826.378,E2 8826.378} C_VEL
LIN {X 0,Y 265.768,Z 840.326,A -85,B 0,C 180,E1 8821.94,E2 8821.94} C_VEL
LIN {X 0,Y 261.301,Z 827.425,A -85,B 0,C 180,E1 8817.046,E2 8817.046} C_VEL
LIN {X 0,Y 257.127,Z 815.929,A -85,B 0,C 180,E1 8812.177,E2 8812.177} C_VEL
LIN {X 0,Y 253.163,Z 805.489,A -85,B 0,C 180,E1 8807.222,E2 8807.222} C_VEL
LIN {X 0,Y 249.665,Z 796.437,A -85,B 0,C 180,E1 8802.384,E2 8802.384} C_VEL
LIN {X 0,Y 246.666,Z 788.764,A -85,B 0,C 180,E1 8797.727,E2 8797.727} C_VEL
LIN {X 0,Y 256.655,Z 789.181,A -85,B 0,C 180,E1 8792.631,E2 8792.631} C_VEL
LIN {X 0,Y 257.027,Z 789.403,A -85,B 0,C 180,E1 8792.423,E2 8792.423} C_VEL
LIN {X 0,Y 259.374,Z 801.278,A -85,B 0,C 180,E1 8789.155,E2 8789.155} C_VEL
LIN {X 0,Y 259.675,Z 803.51,A -85,B 0,C 180,E1 8788.637,E2 8788.637} C_VEL
LIN {X 0,Y 249.333,Z 852.948,A -85,B 0,C 180,E1 8783.706,E2 8783.706} C_VEL
LIN {X 0,Y 242.527,Z 888.168,A -85,B 0,C 180,E1 8780.193,E2 8780.193} C_VEL
LIN {X 0,Y 242.474,Z 894.482,A -85,B 0,C 180,E1 8779.915,E2 8779.915} C_VEL
LIN {X 0,Y 232.131,Z 1038.104,A -85,B 0,C 180,E1 8776.278,E2 8776.278} C_VEL
LIN {X 0,Y 230.616,Z 1063.192,A -85,B 0,C 180,E1 8775.405,E2 8775.405} C_VEL
LIN {X 0,Y 228.393,Z 1081.011,A -85,B 0,C 180,E1 8774.382,E2 8774.382} C_VEL
LIN {X 0,Y 225.37,Z 1096.923,A -85,B 0,C 180,E1 8773.092,E2 8773.092} C_VEL
LIN {X 0,Y 221.428,Z 1112.49,A -85,B 0,C 180,E1 8771.412,E2 8771.412} C_VEL
LIN {X 0,Y 216.533,Z 1127.794,A -85,B 0,C 180,E1 8769.239,E2 8769.239} C_VEL
LIN {X 0,Y 211.111,Z 1141.98,A -85,B 0,C 180,E1 8766.634,E2 8766.634} C_VEL
LIN {X 0,Y 205.566,Z 1154.555,A -85,B 0,C 180,E1 8763.671,E2 8763.671} C_VEL
LIN {X 0,Y 200.055,Z 1165.628,A -85,B 0,C 180,E1 8760.313,E2 8760.313} C_VEL
LIN {X 0,Y 194.421,Z 1175.936,A -85,B 0,C 180,E1 8756.245,E2 8756.245} C_VEL
LIN {X 0,Y 189.352,Z 1184.659,A -85,B 0,C 180,E1 8751.689,E2 8751.689} C_VEL
LIN {X 0,Y 185.31,Z 1191.349,A -85,B 0,C 180,E1 8746.935,E2 8746.935} C_VEL
LIN {X 0,Y 182.177,Z 1196.489,A -85,B 0,C 180,E1 8741.712,E2 8741.712} C_VEL
LIN {X 0,Y 180.135,Z 1200.018,A -85,B 0,C 180,E1 8736.049,E2 8736.049} C_VEL
LIN {X 0,Y 179.328,Z 1201.701,A -85,B 0,C 180,E1 8730.315,E2 8730.315} C_VEL
LIN {X 0,Y 179.662,Z 1201.527,A -85,B 0,C 180,E1 8724.567,E2 8724.567} C_VEL
LIN {X 0,Y 181.202,Z 1199.573,A -85,B 0,C 180,E1 8718.86,E2 8718.86} C_VEL
LIN {X 0,Y 183.851,Z 1196.003,A -85,B 0,C 180,E1 8713.568,E2 8713.568} C_VEL
LIN {X 0,Y 187.698,Z 1190.555,A -85,B 0,C 180,E1 8708.43,E2 8708.43} C_VEL
LIN {X 0,Y 192.747,Z 1183.086,A -85,B 0,C 180,E1 8703.5,E2 8703.5} C_VEL
LIN {X 0,Y 198.154,Z 1174.566,A -85,B 0,C 180,E1 8699.356,E2 8699.356} C_VEL
LIN {X 0,Y 203.941,Z 1164.608,A -85,B 0,C 180,E1 8695.675,E2 8695.675} C_VEL
LIN {X 0,Y 209.886,Z 1153.186,A -85,B 0,C 180,E1 8692.422,E2 8692.422} C_VEL
LIN {X 0,Y 216.076,Z 1139.664,A -85,B 0,C 180,E1 8689.442,E2 8689.442} C_VEL
LIN {X 0,Y 219.881,Z 1129.712,A -85,B 0,C 180,E1 8687.643,E2 8687.643} C_VEL
LIN {X 0,Y 217.561,Z 1129.541,A -85,B 0,C 180,E1 8686.95,E2 8686.95} C_VEL
LIN {X 0,Y 217.097,Z 1129.446,A -85,B 0,C 180,E1 8686.743,E2 8686.743} C_VEL
LIN {X 0,Y 208.756,Z 1148.168,A -85,B 0,C 180,E1 8682.855,E2 8682.855} C_VEL
LIN {X 0,Y 200.48,Z 1166.172,A -85,B 0,C 180,E1 8678.203,E2 8678.203} C_VEL
LIN {X 0,Y 193.378,Z 1181.714,A -85,B 0,C 180,E1 8673.236,E2 8673.236} C_VEL
LIN {X 0,Y 187.237,Z 1195.862,A -85,B 0,C 180,E1 8667.685,E2 8667.685} C_VEL
LIN {X 0,Y 182.133,Z 1209.203,A -85,B 0,C 180,E1 8661.244,E2 8661.244} C_VEL
LIN {X 0,Y 178.798,Z 1220.311,A -85,B 0,C 180,E1 8654.641,E2 8654.641} C_VEL
LIN {X 0,Y 177.051,Z 1229.296,A -85,B 0,C 180,E1 8648.117,E2 8648.117} C_VEL
LIN {X 0,Y 176.468,Z 1236.565,A -85,B 0,C 180,E1 8641.623,E2 8641.623} C_VEL
LIN {X 0,Y 176.513,Z 1241.656,A -85,B 0,C 180,E1 8636.102,E2 8636.102} C_VEL
LIN {X 0,Y 177.252,Z 1246.743,A -85,B 0,C 180,E1 8629.271,E2 8629.271} C_VEL
LIN {X 0,Y 179.821,Z 1251.105,A -85,B 0,C 180,E1 8621.522,E2 8621.522} C_VEL
LIN {X 0,Y 186.362,Z 1254.686,A -85,B 0,C 180,E1 8612.521,E2 8612.521} C_VEL
LIN {X 0,Y 190.351,Z 1255.695,A -85,B 0,C 180,E1 8608.946,E2 8608.946} C_VEL
LIN {X 0,Y 192.259,Z 1256.265,A -85,B 0,C 180,E1 8606.696,E2 8606.696} C_VEL
LIN {X 0,Y 195.591,Z 1257.707,A -85,B 0,C 180,E1 8600.512,E2 8600.512} C_VEL
LIN {X 0,Y 198.3,Z 1258.031,A -85,B 0,C 180,E1 8598.748,E2 8598.748} C_VEL
LIN {X 0,Y 205.252,Z 1258.269,A -85,B 0,C 180,E1 8595.624,E2 8595.624} C_VEL
LIN {X 0,Y 188.569,Z 1261.665,A -85,B 0,C 180,E1 8587.963,E2 8587.963} C_VEL
LIN {X 0,Y 176.972,Z 1263.428,A -85,B 0,C 180,E1 8579.076,E2 8579.076} C_VEL
LIN {X 0,Y 170.839,Z 1263.41,A -85,B 0,C 180,E1 8569.849,E2 8569.849} C_VEL
LIN {X 0,Y 169.094,Z 1261.708,A -85,B 0,C 180,E1 8561.257,E2 8561.257} C_VEL
LIN {X 0,Y 169.582,Z 1258.939,A -85,B 0,C 180,E1 8554.401,E2 8554.401} C_VEL
LIN {X 0,Y 170.095,Z 1255.945,A -85,B 0,C 180,E1 8549.668,E2 8549.668} C_VEL
LIN {X 0,Y 170.019,Z 1251.88,A -85,B 0,C 180,E1 8544.944,E2 8544.944} C_VEL
LIN {X 0,Y 169.897,Z 1245.466,A -85,B 0,C 180,E1 8539.15,E2 8539.15} C_VEL
LIN {X 0,Y 170.646,Z 1236.477,A -85,B 0,C 180,E1 8532.618,E2 8532.618} C_VEL
LIN {X 0,Y 172.619,Z 1226.664,A -85,B 0,C 180,E1 8526.447,E2 8526.447} C_VEL
LIN {X 0,Y 175.592,Z 1217.74,A -85,B 0,C 180,E1 8521.057,E2 8521.057} C_VEL
LIN {X 0,Y 179.556,Z 1207.19,A -85,B 0,C 180,E1 8516.166,E2 8516.166} C_VEL
LIN {X 0,Y 184.313,Z 1195.044,A -85,B 0,C 180,E1 8511.803,E2 8511.803} C_VEL
LIN {X 0,Y 189.241,Z 1181.77,A -85,B 0,C 180,E1 8508.064,E2 8508.064} C_VEL
LIN {X 0,Y 192.621,Z 1172.966,A -85,B 0,C 180,E1 8505.932,E2 8505.932} C_VEL
LIN {X 0,Y 202.65,Z 1150.833,A -85,B 0,C 180,E1 8500.556,E2 8500.556} C_VEL
LIN {X 0,Y 213.368,Z 1127.53,A -85,B 0,C 180,E1 8496.07,E2 8496.07} C_VEL
LIN {X 0,Y 224.354,Z 1103.389,A -85,B 0,C 180,E1 8492.384,E2 8492.384} C_VEL
LIN {X 0,Y 237.373,Z 1074.277,A -85,B 0,C 180,E1 8488.826,E2 8488.826} C_VEL
LIN {X 0,Y 250.658,Z 1043.729,A -85,B 0,C 180,E1 8485.912,E2 8485.912} C_VEL
LIN {X 0,Y 262.471,Z 1014.902,A -85,B 0,C 180,E1 8483.763,E2 8483.763} C_VEL
LIN {X 0,Y 262.297,Z 987.996,A -85,B 0,C 180,E1 8480.065,E2 8480.065} C_VEL
LIN {X 0,Y 263.471,Z 960.385,A -85,B 0,C 180,E1 8476.764,E2 8476.764} C_VEL
LIN {X 0,Y 265.747,Z 931.52,A -85,B 0,C 180,E1 8473.823,E2 8473.823} C_VEL
LIN {X 0,Y 268.934,Z 900.355,A -85,B 0,C 180,E1 8471.202,E2 8471.202} C_VEL
LIN {X 0,Y 271.593,Z 872.511,A -85,B 0,C 180,E1 8469.029,E2 8469.029} C_VEL
LIN {X 0,Y 264.082,Z 855.771,A -85,B 0,C 180,E1 8464.724,E2 8464.724} C_VEL
LIN {X 0,Y 260.587,Z 847.737,A -85,B 0,C 180,E1 8462.419,E2 8462.419} C_VEL
LIN {X 0,Y 256.202,Z 834.684,A -85,B 0,C 180,E1 8457.482,E2 8457.482} C_VEL
LIN {X 0,Y 251.993,Z 822.83,A -85,B 0,C 180,E1 8452.476,E2 8452.476} C_VEL
LIN {X 0,Y 247.998,Z 811.963,A -85,B 0,C 180,E1 8447.327,E2 8447.327} C_VEL
LIN {X 0,Y 244.468,Z 802.726,A -85,B 0,C 180,E1 8442.348,E2 8442.348} C_VEL
LIN {X 0,Y 242.091,Z 796.443,A -85,B 0,C 180,E1 8438.496,E2 8438.496} C_VEL
LIN {X 0,Y 250.512,Z 796.348,A -85,B 0,C 180,E1 8433.956,E2 8433.956} C_VEL
LIN {X 0,Y 252.922,Z 796.545,A -85,B 0,C 180,E1 8432.767,E2 8432.767} C_VEL
LIN {X 0,Y 254.826,Z 807.127,A -85,B 0,C 180,E1 8429.883,E2 8429.883} C_VEL
LIN {X 0,Y 243.893,Z 857.143,A -85,B 0,C 180,E1 8424.867,E2 8424.867} C_VEL
LIN {X 0,Y 237.553,Z 888.956,A -85,B 0,C 180,E1 8421.689,E2 8421.689} C_VEL
LIN {X 0,Y 237.47,Z 895.409,A -85,B 0,C 180,E1 8421.398,E2 8421.398} C_VEL
LIN {X 0,Y 226.786,Z 1038.457,A -85,B 0,C 180,E1 8417.762,E2 8417.762} C_VEL
LIN {X 0,Y 225.163,Z 1064.04,A -85,B 0,C 180,E1 8416.863,E2 8416.863} C_VEL
LIN {X 0,Y 222.861,Z 1081.775,A -85,B 0,C 180,E1 8415.837,E2 8415.837} C_VEL
LIN {X 0,Y 219.647,Z 1098.046,A -85,B 0,C 180,E1 8414.505,E2 8414.505} C_VEL
LIN {X 0,Y 215.544,Z 1113.567,A -85,B 0,C 180,E1 8412.807,E2 8412.807} C_VEL
LIN {X 0,Y 210.45,Z 1128.846,A -85,B 0,C 180,E1 8410.605,E2 8410.605} C_VEL
LIN {X 0,Y 204.8,Z 1143.016,A -85,B 0,C 180,E1 8407.959,E2 8407.959} C_VEL
LIN {X 0,Y 199.012,Z 1155.578,A -85,B 0,C 180,E1 8404.938,E2 8404.938} C_VEL
LIN {X 0,Y 193.245,Z 1166.636,A -85,B 0,C 180,E1 8401.501,E2 8401.501} C_VEL
LIN {X 0,Y 187.333,Z 1176.935,A -85,B 0,C 180,E1 8397.319,E2 8397.319} C_VEL
LIN {X 0,Y 181.996,Z 1185.65,A -85,B 0,C 180,E1 8392.613,E2 8392.613} C_VEL
LIN {X 0,Y 177.727,Z 1192.329,A -85,B 0,C 180,E1 8387.681,E2 8387.681} C_VEL
LIN {X 0,Y 174.408,Z 1197.461,A -85,B 0,C 180,E1 8382.242,E2 8382.242} C_VEL
LIN {X 0,Y 172.24,Z 1200.983,A -85,B 0,C 180,E1 8376.328,E2 8376.328} C_VEL
LIN {X 0,Y 171.385,Z 1202.656,A -85,B 0,C 180,E1 8370.33,E2 8370.33} C_VEL
LIN {X 0,Y 171.75,Z 1202.476,A -85,B 0,C 180,E1 8364.316,E2 8364.316} C_VEL
LIN {X 0,Y 173.402,Z 1200.515,A -85,B 0,C 180,E1 8358.352,E2 8358.352} C_VEL
LIN {X 0,Y 176.229,Z 1196.937,A -85,B 0,C 180,E1 8352.836,E2 8352.836} C_VEL
LIN {X 0,Y 180.316,Z 1191.478,A -85,B 0,C 180,E1 8347.5,E2 8347.5} C_VEL
LIN {X 0,Y 185.655,Z 1184,A -85,B 0,C 180,E1 8342.404,E2 8342.404} C_VEL
LIN {X 0,Y 191.348,Z 1175.469,A -85,B 0,C 180,E1 8338.14,E2 8338.14} C_VEL
LIN {X 0,Y 197.418,Z 1165.493,A -85,B 0,C 180,E1 8334.372,E2 8334.372} C_VEL
LIN {X 0,Y 203.636,Z 1154.057,A -85,B 0,C 180,E1 8331.056,E2 8331.056} C_VEL
LIN {X 0,Y 210.093,Z 1140.516,A -85,B 0,C 180,E1 8328.031,E2 8328.031} C_VEL
LIN {X 0,Y 211.114,Z 1137.759,A -85,B 0,C 180,E1 8327.454,E2 8327.454} C_VEL
LIN {X 0,Y 207.688,Z 1138.425,A -85,B 0,C 180,E1 8326.633,E2 8326.633} C_VEL
LIN {X 0,Y 205.948,Z 1138.128,A -85,B 0,C 180,E1 8325.935,E2 8325.935} C_VEL
LIN {X 0,Y 197.588,Z 1156.075,A -85,B 0,C 180,E1 8321.717,E2 8321.717} C_VEL
LIN {X 0,Y 189.779,Z 1172.576,A -85,B 0,C 180,E1 8316.916,E2 8316.916} C_VEL
LIN {X 0,Y 182.305,Z 1188.828,A -85,B 0,C 180,E1 8311.035,E2 8311.035} C_VEL
LIN {X 0,Y 176.474,Z 1202.676,A -85,B 0,C 180,E1 8304.789,E2 8304.789} C_VEL
LIN {X 0,Y 172.319,Z 1214.488,A -85,B 0,C 180,E1 8298.261,E2 8298.261} C_VEL
LIN {X 0,Y 169.801,Z 1224.376,A -85,B 0,C 180,E1 8291.55,E2 8291.55} C_VEL
LIN {X 0,Y 168.657,Z 1232.615,A -85,B 0,C 180,E1 8284.761,E2 8284.761} C_VEL
LIN {X 0,Y 168.474,Z 1238.762,A -85,B 0,C 180,E1 8278.64,E2 8278.64} C_VEL
LIN {X 0,Y 168.87,Z 1244.313,A -85,B 0,C 180,E1 8271.83,E2 8271.83} C_VEL
LIN {X 0,Y 170.557,Z 1249.088,A -85,B 0,C 180,E1 8264.355,E2 8264.355} C_VEL
LIN {X 0,Y 175.751,Z 1253.562,A -85,B 0,C 180,E1 8255.102,E2 8255.102} C_VEL
LIN {X 0,Y 186.12,Z 1256.689,A -85,B 0,C 180,E1 8245.661,E2 8245.661} C_VEL
LIN {X 0,Y 198.3,Z 1258.031,A -85,B 0,C 180,E1 8238.748,E2 8238.748} C_VEL
LIN {X 0,Y 199.049,Z 1258.235,A -85,B 0,C 180,E1 8237.888,E2 8237.888} C_VEL
LIN {X 0,Y 197.997,Z 1258.672,A -85,B 0,C 180,E1 8236.579,E2 8236.579} C_VEL
LIN {X 0,Y 194.624,Z 1259.293,A -85,B 0,C 180,E1 8235.033,E2 8235.033} C_VEL
LIN {X 0,Y 187.73,Z 1260.37,A -85,B 0,C 180,E1 8232.384,E2 8232.384} C_VEL
LIN {X 0,Y 173.455,Z 1262.281,A -85,B 0,C 180,E1 8223.605,E2 8223.605} C_VEL
LIN {X 0,Y 164.875,Z 1262.517,A -85,B 0,C 180,E1 8213.979,E2 8213.979} C_VEL
LIN {X 0,Y 161.489,Z 1260.978,A -85,B 0,C 180,E1 8204.344,E2 8204.344} C_VEL
LIN {X 0,Y 161.529,Z 1258.181,A -85,B 0,C 180,E1 8196.402,E2 8196.402} C_VEL
LIN {X 0,Y 162.202,Z 1255.152,A -85,B 0,C 180,E1 8191.064,E2 8191.064} C_VEL
LIN {X 0,Y 162.265,Z 1251.545,A -85,B 0,C 180,E1 8186.472,E2 8186.472} C_VEL
LIN {X 0,Y 162.024,Z 1245.765,A -85,B 0,C 180,E1 8180.772,E2 8180.772} C_VEL
LIN {X 0,Y 162.452,Z 1237.592,A -85,B 0,C 180,E1 8174.292,E2 8174.292} C_VEL
LIN {X 0,Y 163.386,Z 1231.386,A -85,B 0,C 180,E1 8169.963,E2 8169.963} C_VEL
LIN {X 0,Y 165.61,Z 1223.95,A -85,B 0,C 180,E1 8164.106,E2 8164.106} C_VEL
LIN {X 0,Y 169.118,Z 1214.743,A -85,B 0,C 180,E1 8158.654,E2 8158.654} C_VEL
LIN {X 0,Y 173.711,Z 1203.73,A -85,B 0,C 180,E1 8153.645,E2 8153.645} C_VEL
LIN {X 0,Y 178.835,Z 1191.557,A -85,B 0,C 180,E1 8149.362,E2 8149.362} C_VEL
LIN {X 0,Y 184.084,Z 1178.274,A -85,B 0,C 180,E1 8145.742,E2 8145.742} C_VEL
LIN {X 0,Y 189.428,Z 1163.397,A -85,B 0,C 180,E1 8142.586,E2 8142.586} C_VEL
LIN {X 0,Y 191.281,Z 1158.905,A -85,B 0,C 180,E1 8141.632,E2 8141.632} C_VEL
LIN {X 0,Y 201.634,Z 1137,A -85,B 0,C 180,E1 8136.872,E2 8136.872} C_VEL
LIN {X 0,Y 212.834,Z 1113.207,A -85,B 0,C 180,E1 8132.769,E2 8132.769} C_VEL
LIN {X 0,Y 227.197,Z 1081.879,A -85,B 0,C 180,E1 8128.607,E2 8128.607} C_VEL
LIN {X 0,Y 241.253,Z 1050.484,A -85,B 0,C 180,E1 8125.385,E2 8125.385} C_VEL
LIN {X 0,Y 254.561,Z 1019.331,A -85,B 0,C 180,E1 8122.924,E2 8122.924} C_VEL
LIN {X 0,Y 255.903,Z 1015.61,A -85,B 0,C 180,E1 8122.636,E2 8122.636} C_VEL
LIN {X 0,Y 256.185,Z 988.183,A -85,B 0,C 180,E1 8118.784,E2 8118.784} C_VEL
LIN {X 0,Y 257.852,Z 959.159,A -85,B 0,C 180,E1 8115.289,E2 8115.289} C_VEL
LIN {X 0,Y 260.507,Z 931.196,A -85,B 0,C 180,E1 8112.412,E2 8112.412} C_VEL
LIN {X 0,Y 264.369,Z 897.114,A -85,B 0,C 180,E1 8109.544,E2 8109.544} C_VEL
LIN {X 0,Y 266.454,Z 876.518,A -85,B 0,C 180,E1 8107.902,E2 8107.902} C_VEL
LIN {X 0,Y 259.383,Z 860.645,A -85,B 0,C 180,E1 8103.702,E2 8103.702} C_VEL
LIN {X 0,Y 254.241,Z 849.326,A -85,B 0,C 180,E1 8100.338,E2 8100.338} C_VEL
LIN {X 0,Y 250.895,Z 841.446,A -85,B 0,C 180,E1 8097.716,E2 8097.716} C_VEL
LIN {X 0,Y 246.856,Z 829.763,A -85,B 0,C 180,E1 8092.787,E2 8092.787} C_VEL
LIN {X 0,Y 243.137,Z 819.41,A -85,B 0,C 180,E1 8087.893,E2 8087.893} C_VEL
LIN {X 0,Y 239.956,Z 810.698,A -85,B 0,C 180,E1 8083.29,E2 8083.29} C_VEL
LIN {X 0,Y 237.612,Z 804.113,A -85,B 0,C 180,E1 8079.3,E2 8079.3} C_VEL
LIN {X 0,Y 246.615,Z 803.685,A -85,B 0,C 180,E1 8074.289,E2 8074.289} C_VEL
LIN {X 0,Y 248.956,Z 804.013,A -85,B 0,C 180,E1 8073.07,E2 8073.07} C_VEL
LIN {X 0,Y 250.013,Z 811.138,A -85,B 0,C 180,E1 8071.139,E2 8071.139} C_VEL
LIN {X 0,Y 238.761,Z 860.801,A -85,B 0,C 180,E1 8066.153,E2 8066.153} C_VEL
LIN {X 0,Y 232.749,Z 889.909,A -85,B 0,C 180,E1 8063.238,E2 8063.238} C_VEL
LIN {X 0,Y 232.631,Z 896.345,A -85,B 0,C 180,E1 8062.944,E2 8062.944} C_VEL
LIN {X 0,Y 221.6,Z 1038.811,A -85,B 0,C 180,E1 8059.316,E2 8059.316} C_VEL
LIN {X 0,Y 219.862,Z 1064.896,A -85,B 0,C 180,E1 8058.393,E2 8058.393} C_VEL
LIN {X 0,Y 217.463,Z 1082.643,A -85,B 0,C 180,E1 8057.358,E2 8057.358} C_VEL
LIN {X 0,Y 214.064,Z 1099.17,A -85,B 0,C 180,E1 8055.993,E2 8055.993} C_VEL
LIN {X 0,Y 209.794,Z 1114.641,A -85,B 0,C 180,E1 8054.279,E2 8054.279} C_VEL
LIN {X 0,Y 204.493,Z 1129.899,A -85,B 0,C 180,E1 8052.051,E2 8052.051} C_VEL
LIN {X 0,Y 198.605,Z 1144.054,A -85,B 0,C 180,E1 8049.366,E2 8049.366} C_VEL
LIN {X 0,Y 192.561,Z 1156.6,A -85,B 0,C 180,E1 8046.29,E2 8046.29} C_VEL
LIN {X 0,Y 186.523,Z 1167.643,A -85,B 0,C 180,E1 8042.775,E2 8042.775} C_VEL
LIN {X 0,Y 180.316,Z 1177.934,A -85,B 0,C 180,E1 8038.477,E2 8038.477} C_VEL
LIN {X 0,Y 174.693,Z 1186.64,A -85,B 0,C 180,E1 8033.614,E2 8033.614} C_VEL
LIN {X 0,Y 170.176,Z 1193.308,A -85,B 0,C 180,E1 8028.494,E2 8028.494} C_VEL
LIN {X 0,Y 166.654,Z 1198.433,A -85,B 0,C 180,E1 8022.821,E2 8022.821} C_VEL
LIN {X 0,Y 164.348,Z 1201.948,A -85,B 0,C 180,E1 8016.633,E2 8016.633} C_VEL
LIN {X 0,Y 163.441,Z 1203.611,A -85,B 0,C 180,E1 8010.346,E2 8010.346} C_VEL
LIN {X 0,Y 163.842,Z 1203.424,A -85,B 0,C 180,E1 8004.04,E2 8004.04} C_VEL
LIN {X 0,Y 165.619,Z 1201.456,A -85,B 0,C 180,E1 7997.796,E2 7997.796} C_VEL
LIN {X 0,Y 168.64,Z 1197.871,A -85,B 0,C 180,E1 7992.038,E2 7992.038} C_VEL
LIN {X 0,Y 172.986,Z 1192.401,A -85,B 0,C 180,E1 7986.49,E2 7986.49} C_VEL
LIN {X 0,Y 178.635,Z 1184.914,A -85,B 0,C 180,E1 7981.22,E2 7981.22} C_VEL
LIN {X 0,Y 184.633,Z 1176.372,A -85,B 0,C 180,E1 7976.836,E2 7976.836} C_VEL
LIN {X 0,Y 191.003,Z 1166.379,A -85,B 0,C 180,E1 7972.981,E2 7972.981} C_VEL
LIN {X 0,Y 197.508,Z 1154.928,A -85,B 0,C 180,E1 7969.604,E2 7969.604} C_VEL
LIN {X 0,Y 202.627,Z 1144.788,A -85,B 0,C 180,E1 7967.226,E2 7967.226} C_VEL
LIN {X 0,Y 197.962,Z 1146.243,A -85,B 0,C 180,E1 7966.244,E2 7966.244} C_VEL
LIN {X 0,Y 195.379,Z 1146.181,A -85,B 0,C 180,E1 7965.346,E2 7965.346} C_VEL
LIN {X 0,Y 194.878,Z 1146.023,A -85,B 0,C 180,E1 7965.077,E2 7965.077} C_VEL
LIN {X 0,Y 185.997,Z 1164.409,A -85,B 0,C 180,E1 7960.173,E2 7960.173} C_VEL
LIN {X 0,Y 177.966,Z 1181.07,A -85,B 0,C 180,E1 7954.574,E2 7954.574} C_VEL
LIN {X 0,Y 171.132,Z 1196.12,A -85,B 0,C 180,E1 7948.247,E2 7948.247} C_VEL
LIN {X 0,Y 166.05,Z 1208.946,A -85,B 0,C 180,E1 7941.551,E2 7941.551} C_VEL
LIN {X 0,Y 162.72,Z 1219.793,A -85,B 0,C 180,E1 7934.592,E2 7934.592} C_VEL
LIN {X 0,Y 160.997,Z 1228.858,A -85,B 0,C 180,E1 7927.494,E2 7927.494} C_VEL
LIN {X 0,Y 160.514,Z 1236.074,A -85,B 0,C 180,E1 7920.714,E2 7920.714} C_VEL
LIN {X 0,Y 160.695,Z 1241.906,A -85,B 0,C 180,E1 7913.928,E2 7913.928} C_VEL
LIN {X 0,Y 161.807,Z 1246.909,A -85,B 0,C 180,E1 7906.783,E2 7906.783} C_VEL
LIN {X 0,Y 166.074,Z 1252.191,A -85,B 0,C 180,E1 7897.109,E2 7897.109} C_VEL
LIN {X 0,Y 175.357,Z 1256.196,A -85,B 0,C 180,E1 7887.201,E2 7887.201} C_VEL
LIN {X 0,Y 190.235,Z 1258.633,A -85,B 0,C 180,E1 7878.124,E2 7878.124} C_VEL
LIN {X 0,Y 195.504,Z 1259.045,A -85,B 0,C 180,E1 7875.732,E2 7875.732} C_VEL
LIN {X 0,Y 187.73,Z 1260.37,A -85,B 0,C 180,E1 7872.384,E2 7872.384} C_VEL
LIN {X 0,Y 182.491,Z 1261.001,A -85,B 0,C 180,E1 7870.391,E2 7870.391} C_VEL
LIN {X 0,Y 168.41,Z 1261.523,A -85,B 0,C 180,E1 7865.699,E2 7865.699} C_VEL
LIN {X 0,Y 164.822,Z 1261.536,A -85,B 0,C 180,E1 7863.554,E2 7863.554} C_VEL
LIN {X 0,Y 156.472,Z 1261.129,A -85,B 0,C 180,E1 7853.345,E2 7853.345} C_VEL
LIN {X 0,Y 153.563,Z 1259.082,A -85,B 0,C 180,E1 7843.562,E2 7843.562} C_VEL
LIN {X 0,Y 153.807,Z 1256.08,A -85,B 0,C 180,E1 7835.929,E2 7835.929} C_VEL
LIN {X 0,Y 154.444,Z 1253.082,A -85,B 0,C 180,E1 7830.747,E2 7830.747} C_VEL
LIN {X 0,Y 154.413,Z 1249.228,A -85,B 0,C 180,E1 7825.92,E2 7825.92} C_VEL
LIN {X 0,Y 154.181,Z 1243.083,A -85,B 0,C 180,E1 7819.921,E2 7819.921} C_VEL
LIN {X 0,Y 154.808,Z 1234.256,A -85,B 0,C 180,E1 7812.925,E2 7812.925} C_VEL
LIN {X 0,Y 156.705,Z 1226.921,A -85,B 0,C 180,E1 7805.846,E2 7805.846} C_VEL
LIN {X 0,Y 159.901,Z 1218.675,A -85,B 0,C 180,E1 7799.989,E2 7799.989} C_VEL
LIN {X 0,Y 164.239,Z 1208.825,A -85,B 0,C 180,E1 7794.666,E2 7794.666} C_VEL
LIN {X 0,Y 169.429,Z 1197.543,A -85,B 0,C 180,E1 7789.971,E2 7789.971} C_VEL
LIN {X 0,Y 175.074,Z 1184.733,A -85,B 0,C 180,E1 7785.839,E2 7785.839} C_VEL
LIN {X 0,Y 180.726,Z 1170.797,A -85,B 0,C 180,E1 7782.395,E2 7782.395} C_VEL
LIN {X 0,Y 186.065,Z 1155.955,A -85,B 0,C 180,E1 7779.55,E2 7779.55} C_VEL
LIN {X 0,Y 188.853,Z 1148.134,A -85,B 0,C 180,E1 7778.277,E2 7778.277} C_VEL
LIN {X 0,Y 200.377,Z 1124.345,A -85,B 0,C 180,E1 7773.565,E2 7773.565} C_VEL
LIN {X 0,Y 211.988,Z 1099.982,A -85,B 0,C 180,E1 7769.796,E2 7769.796} C_VEL
LIN {X 0,Y 226.045,Z 1069.818,A -85,B 0,C 180,E1 7766.12,E2 7766.12} C_VEL
LIN {X 0,Y 239.902,Z 1039.162,A -85,B 0,C 180,E1 7763.227,E2 7763.227} C_VEL
LIN {X 0,Y 249.383,Z 1016.821,A -85,B 0,C 180,E1 7761.546,E2 7761.546} C_VEL
LIN {X 0,Y 249.912,Z 991.763,A -85,B 0,C 180,E1 7757.943,E2 7757.943} C_VEL
LIN {X 0,Y 251.864,Z 963.475,A -85,B 0,C 180,E1 7754.396,E2 7754.396} C_VEL
LIN {X 0,Y 254.589,Z 936.894,A -85,B 0,C 180,E1 7751.555,E2 7751.555} C_VEL
LIN {X 0,Y 258.465,Z 905.919,A -85,B 0,C 180,E1 7748.804,E2 7748.804} C_VEL
LIN {X 0,Y 261.337,Z 880.67,A -85,B 0,C 180,E1 7746.757,E2 7746.757} C_VEL
LIN {X 0,Y 254.643,Z 865.295,A -85,B 0,C 180,E1 7742.588,E2 7742.588} C_VEL
LIN {X 0,Y 248.803,Z 852.219,A -85,B 0,C 180,E1 7738.561,E2 7738.561} C_VEL
LIN {X 0,Y 242.262,Z 837.847,A -85,B 0,C 180,E1 7733.483,E2 7733.483} C_VEL
LIN {X 0,Y 240.248,Z 832.392,A -85,B 0,C 180,E1 7731.142,E2 7731.142} C_VEL
LIN {X 0,Y 236.47,Z 821.698,A -85,B 0,C 180,E1 7725.803,E2 7725.803} C_VEL
LIN {X 0,Y 233.209,Z 812.693,A -85,B 0,C 180,E1 7720.723,E2 7720.723} C_VEL
LIN {X 0,Y 233.094,Z 812.035,A -85,B 0,C 180,E1 7720.191,E2 7720.191} C_VEL
LIN {X 0,Y 241.015,Z 811.123,A -85,B 0,C 180,E1 7715.489,E2 7715.489} C_VEL
LIN {X 0,Y 244.947,Z 811.342,A -85,B 0,C 180,E1 7713.436,E2 7713.436} C_VEL
LIN {X 0,Y 245.335,Z 815.107,A -85,B 0,C 180,E1 7712.447,E2 7712.447} C_VEL
LIN {X 0,Y 233.671,Z 864.994,A -85,B 0,C 180,E1 7707.448,E2 7707.448} C_VEL
LIN {X 0,Y 228.122,Z 890.86,A -85,B 0,C 180,E1 7704.851,E2 7704.851} C_VEL
LIN {X 0,Y 227.977,Z 897.191,A -85,B 0,C 180,E1 7704.556,E2 7704.556} C_VEL
LIN {X 0,Y 216.584,Z 1039.159,A -85,B 0,C 180,E1 7700.944,E2 7700.944} C_VEL
LIN {X 0,Y 214.733,Z 1065.702,A -85,B 0,C 180,E1 7699.998,E2 7699.998} C_VEL
LIN {X 0,Y 212.263,Z 1083.305,A -85,B 0,C 180,E1 7698.97,E2 7698.97} C_VEL
LIN {X 0,Y 208.927,Z 1099.059,A -85,B 0,C 180,E1 7697.675,E2 7697.675} C_VEL
LIN {X 0,Y 204.488,Z 1114.817,A -85,B 0,C 180,E1 7695.948,E2 7695.948} C_VEL
LIN {X 0,Y 199.249,Z 1129.529,A -85,B 0,C 180,E1 7693.824,E2 7693.824} C_VEL
LIN {X 0,Y 193.081,Z 1143.912,A -85,B 0,C 180,E1 7691.117,E2 7691.117} C_VEL
LIN {X 0,Y 186.731,Z 1156.645,A -85,B 0,C 180,E1 7688.003,E2 7688.003} C_VEL
LIN {X 0,Y 180.368,Z 1167.902,A -85,B 0,C 180,E1 7684.428,E2 7684.428} C_VEL
LIN {X 0,Y 173.784,Z 1178.318,A -85,B 0,C 180,E1 7680.032,E2 7680.032} C_VEL
LIN {X 0,Y 167.782,Z 1187.134,A -85,B 0,C 180,E1 7675.026,E2 7675.026} C_VEL
LIN {X 0,Y 162.928,Z 1193.938,A -85,B 0,C 180,E1 7669.721,E2 7669.721} C_VEL
LIN {X 0,Y 159.103,Z 1199.16,A -85,B 0,C 180,E1 7663.811,E2 7663.811} C_VEL
LIN {X 0,Y 156.557,Z 1202.759,A -85,B 0,C 180,E1 7657.334,E2 7657.334} C_VEL
LIN {X 0,Y 155.516,Z 1204.529,A -85,B 0,C 180,E1 7650.732,E2 7650.732} C_VEL
LIN {X 0,Y 155.876,Z 1204.435,A -85,B 0,C 180,E1 7644.104,E2 7644.104} C_VEL
LIN {X 0,Y 157.722,Z 1202.53,A -85,B 0,C 180,E1 7637.502,E2 7637.502} C_VEL
LIN {X 0,Y 161.086,Z 1198.805,A -85,B 0,C 180,E1 7631.164,E2 7631.164} C_VEL
LIN {X 0,Y 165.714,Z 1193.323,A -85,B 0,C 180,E1 7625.392,E2 7625.392} C_VEL
LIN {X 0,Y 171.698,Z 1185.827,A -85,B 0,C 180,E1 7619.941,E2 7619.941} C_VEL
LIN {X 0,Y 178.022,Z 1177.275,A -85,B 0,C 180,E1 7615.434,E2 7615.434} C_VEL
LIN {X 0,Y 184.709,Z 1167.265,A -85,B 0,C 180,E1 7611.494,E2 7611.494} C_VEL
LIN {X 0,Y 191.516,Z 1155.798,A -85,B 0,C 180,E1 7608.061,E2 7608.061} C_VEL
LIN {X 0,Y 193.389,Z 1152.271,A -85,B 0,C 180,E1 7607.131,E2 7607.131} C_VEL
LIN {X 0,Y 191.578,Z 1152.259,A -85,B 0,C 180,E1 7606.509,E2 7606.509} C_VEL
LIN {X 0,Y 186.807,Z 1153.621,A -85,B 0,C 180,E1 7605.389,E2 7605.389} C_VEL
LIN {X 0,Y 184.064,Z 1153.455,A -85,B 0,C 180,E1 7604.271,E2 7604.271} C_VEL
LIN {X 0,Y 183.743,Z 1153.596,A -85,B 0,C 180,E1 7604.079,E2 7604.079} C_VEL
LIN {X 0,Y 175.156,Z 1170.829,A -85,B 0,C 180,E1 7598.899,E2 7598.899} C_VEL
LIN {X 0,Y 167.446,Z 1186.631,A -85,B 0,C 180,E1 7592.916,E2 7592.916} C_VEL
LIN {X 0,Y 161.065,Z 1200.868,A -85,B 0,C 180,E1 7586.153,E2 7586.153} C_VEL
LIN {X 0,Y 156.537,Z 1212.963,A -85,B 0,C 180,E1 7579.012,E2 7579.012} C_VEL
LIN {X 0,Y 153.741,Z 1223.689,A -85,B 0,C 180,E1 7571.251,E2 7571.251} C_VEL
LIN {X 0,Y 152.653,Z 1232.221,A -85,B 0,C 180,E1 7563.756,E2 7563.756} C_VEL
LIN {X 0,Y 152.581,Z 1238.489,A -85,B 0,C 180,E1 7556.995,E2 7556.995} C_VEL
LIN {X 0,Y 153.147,Z 1243.698,A -85,B 0,C 180,E1 7550.227,E2 7550.227} C_VEL
LIN {X 0,Y 155.836,Z 1249.504,A -85,B 0,C 180,E1 7540.899,E2 7540.899} C_VEL
LIN {X 0,Y 163.351,Z 1254.649,A -85,B 0,C 180,E1 7530.277,E2 7530.277} C_VEL
LIN {X 0,Y 177.816,Z 1258.421,A -85,B 0,C 180,E1 7519.709,E2 7519.709} C_VEL
LIN {X 0,Y 185.614,Z 1259.446,A -85,B 0,C 180,E1 7515.768,E2 7515.768} C_VEL
LIN {X 0,Y 169.746,Z 1261.24,A -85,B 0,C 180,E1 7507.358,E2 7507.358} C_VEL
LIN {X 0,Y 164.822,Z 1261.536,A -85,B 0,C 180,E1 7503.554,E2 7503.554} C_VEL
LIN {X 0,Y 160.916,Z 1261.497,A -85,B 0,C 180,E1 7500.969,E2 7500.969} C_VEL
LIN {X 0,Y 149.843,Z 1259.951,A -85,B 0,C 180,E1 7494.541,E2 7494.541} C_VEL
LIN {X 0,Y 147.887,Z 1259.372,A -85,B 0,C 180,E1 7492.1,E2 7492.1} C_VEL
LIN {X 0,Y 145.676,Z 1256.674,A -85,B 0,C 180,E1 7481.888,E2 7481.888} C_VEL
LIN {X 0,Y 146.26,Z 1253.275,A -85,B 0,C 180,E1 7474.318,E2 7474.318} C_VEL
LIN {X 0,Y 146.726,Z 1250.289,A -85,B 0,C 180,E1 7469.615,E2 7469.615} C_VEL
LIN {X 0,Y 146.512,Z 1246.012,A -85,B 0,C 180,E1 7464.523,E2 7464.523} C_VEL
LIN {X 0,Y 146.407,Z 1238.66,A -85,B 0,C 180,E1 7457.588,E2 7457.588} C_VEL
LIN {X 0,Y 146.682,Z 1234.824,A -85,B 0,C 180,E1 7454.183,E2 7454.183} C_VEL
LIN {X 0,Y 148.058,Z 1228.967,A -85,B 0,C 180,E1 7447.366,E2 7447.366} C_VEL
LIN {X 0,Y 150.99,Z 1221.527,A -85,B 0,C 180,E1 7441.097,E2 7441.097} C_VEL
LIN {X 0,Y 155.443,Z 1211.97,A -85,B 0,C 180,E1 7435.082,E2 7435.082} C_VEL
LIN {X 0,Y 160.924,Z 1200.966,A -85,B 0,C 180,E1 7429.841,E2 7429.841} C_VEL
LIN {X 0,Y 166.767,Z 1188.902,A -85,B 0,C 180,E1 7425.46,E2 7425.46} C_VEL
LIN {X 0,Y 172.964,Z 1175.193,A -85,B 0,C 180,E1 7421.668,E2 7421.668} C_VEL
LIN {X 0,Y 178.914,Z 1160.428,A -85,B 0,C 180,E1 7418.526,E2 7418.526} C_VEL
LIN {X 0,Y 184.201,Z 1145.103,A -85,B 0,C 180,E1 7416.029,E2 7416.029} C_VEL
LIN {X 0,Y 186.944,Z 1136.894,A -85,B 0,C 180,E1 7414.911,E2 7414.911} C_VEL
LIN {X 0,Y 199.717,Z 1111.089,A -85,B 0,C 180,E1 7410.283,E2 7410.283} C_VEL
LIN {X 0,Y 215.156,Z 1078.909,A -85,B 0,C 180,E1 7405.951,E2 7405.951} C_VEL
LIN {X 0,Y 230.226,Z 1046.566,A -85,B 0,C 180,E1 7402.656,E2 7402.656} C_VEL
LIN {X 0,Y 242.903,Z 1017.618,A -85,B 0,C 180,E1 7400.355,E2 7400.355} C_VEL
LIN {X 0,Y 243.883,Z 991.56,A -85,B 0,C 180,E1 7396.543,E2 7396.543} C_VEL
LIN {X 0,Y 246.462,Z 961.765,A -85,B 0,C 180,E1 7392.774,E2 7392.774} C_VEL
LIN {X 0,Y 249.663,Z 934.648,A -85,B 0,C 180,E1 7389.886,E2 7389.886} C_VEL
LIN {X 0,Y 254.475,Z 899.767,A -85,B 0,C 180,E1 7386.826,E2 7386.826} C_VEL
LIN {X 0,Y 256.287,Z 884.909,A -85,B 0,C 180,E1 7385.597,E2 7385.597} C_VEL
LIN {X 0,Y 250.003,Z 870.164,A -85,B 0,C 180,E1 7381.521,E2 7381.521} C_VEL
LIN {X 0,Y 243.007,Z 854.16,A -85,B 0,C 180,E1 7376.402,E2 7376.402} C_VEL
LIN {X 0,Y 236.519,Z 839.711,A -85,B 0,C 180,E1 7370.94,E2 7370.94} C_VEL
LIN {X 0,Y 230.495,Z 825.865,A -85,B 0,C 180,E1 7364.656,E2 7364.656} C_VEL
LIN {X 0,Y 228.477,Z 820.029,A -85,B 0,C 180,E1 7361.236,E2 7361.236} C_VEL
LIN {X 0,Y 236.413,Z 818.652,A -85,B 0,C 180,E1 7356.309,E2 7356.309} C_VEL
LIN {X 0,Y 240.899,Z 818.6,A -85,B 0,C 180,E1 7353.853,E2 7353.853} C_VEL
LIN {X 0,Y 228.899,Z 868.361,A -85,B 0,C 180,E1 7348.882,E2 7348.882} C_VEL
LIN {X 0,Y 223.684,Z 891.857,A -85,B 0,C 180,E1 7346.527,E2 7346.527} C_VEL
LIN {X 0,Y 223.499,Z 898.164,A -85,B 0,C 180,E1 7346.231,E2 7346.231} C_VEL
LIN {X 0,Y 211.752,Z 1039.506,A -85,B 0,C 180,E1 7342.647,E2 7342.647} C_VEL
LIN {X 0,Y 209.763,Z 1066.641,A -85,B 0,C 180,E1 7341.675,E2 7341.675} C_VEL
LIN {X 0,Y 207.181,Z 1084.272,A -85,B 0,C 180,E1 7340.639,E2 7340.639} C_VEL
LIN {X 0,Y 203.672,Z 1100.179,A -85,B 0,C 180,E1 7339.324,E2 7339.324} C_VEL
LIN {X 0,Y 199.055,Z 1115.899,A -85,B 0,C 180,E1 7337.589,E2 7337.589} C_VEL
LIN {X 0,Y 193.606,Z 1130.582,A -85,B 0,C 180,E1 7335.449,E2 7335.449} C_VEL
LIN {X 0,Y 187.178,Z 1144.949,A -85,B 0,C 180,E1 7332.714,E2 7332.714} C_VEL
LIN {X 0,Y 180.545,Z 1157.669,A -85,B 0,C 180,E1 7329.554,E2 7329.554} C_VEL
LIN {X 0,Y 173.88,Z 1168.911,A -85,B 0,C 180,E1 7325.906,E2 7325.906} C_VEL
LIN {X 0,Y 167.393,Z 1178.703,A -85,B 0,C 180,E1 7321.706,E2 7321.706} C_VEL
LIN {X 0,Y 160.983,Z 1187.627,A -85,B 0,C 180,E1 7316.559,E2 7316.559} C_VEL
LIN {X 0,Y 155.759,Z 1194.535,A -85,B 0,C 180,E1 7311.063,E2 7311.063} C_VEL
LIN {X 0,Y 151.602,Z 1199.888,A -85,B 0,C 180,E1 7304.9,E2 7304.9} C_VEL
LIN {X 0,Y 148.792,Z 1203.57,A -85,B 0,C 180,E1 7298.107,E2 7298.107} C_VEL
LIN {X 0,Y 147.596,Z 1205.421,A -85,B 0,C 180,E1 7291.159,E2 7291.159} C_VEL
LIN {X 0,Y 147.855,Z 1205.509,A -85,B 0,C 180,E1 7284.562,E2 7284.562} C_VEL
LIN {X 0,Y 149.645,Z 1203.793,A -85,B 0,C 180,E1 7277.649,E2 7277.649} C_VEL
LIN {X 0,Y 153.084,Z 1200.228,A -85,B 0,C 180,E1 7270.933,E2 7270.933} C_VEL
LIN {X 0,Y 157.856,Z 1195.021,A -85,B 0,C 180,E1 7264.883,E2 7264.883} C_VEL
LIN {X 0,Y 163.763,Z 1188.076,A -85,B 0,C 180,E1 7259.419,E2 7259.419} C_VEL
LIN {X 0,Y 170.579,Z 1179.408,A -85,B 0,C 180,E1 7254.522,E2 7254.522} C_VEL
LIN {X 0,Y 178.025,Z 1168.96,A -85,B 0,C 180,E1 7250.182,E2 7250.182} C_VEL
LIN {X 0,Y 184.153,Z 1159.095,A -85,B 0,C 180,E1 7247.025,E2 7247.025} C_VEL
LIN {X 0,Y 179.497,Z 1159.526,A -85,B 0,C 180,E1 7245.482,E2 7245.482} C_VEL
LIN {X 0,Y 175.006,Z 1160.543,A -85,B 0,C 180,E1 7244.191,E2 7244.191} C_VEL
LIN {X 0,Y 172.794,Z 1160.297,A -85,B 0,C 180,E1 7243.065,E2 7243.065} C_VEL
LIN {X 0,Y 164.374,Z 1176.733,A -85,B 0,C 180,E1 7237.467,E2 7237.467} C_VEL
LIN {X 0,Y 157.028,Z 1191.714,A -85,B 0,C 180,E1 7231.049,E2 7231.049} C_VEL
LIN {X 0,Y 151.159,Z 1205.26,A -85,B 0,C 180,E1 7223.798,E2 7223.798} C_VEL
LIN {X 0,Y 147.243,Z 1216.786,A -85,B 0,C 180,E1 7216.166,E2 7216.166} C_VEL
LIN {X 0,Y 145.251,Z 1225.98,A -85,B 0,C 180,E1 7208.711,E2 7208.711} C_VEL
LIN {X 0,Y 144.613,Z 1233.766,A -85,B 0,C 180,E1 7201.189,E2 7201.189} C_VEL
LIN {X 0,Y 144.784,Z 1239.833,A -85,B 0,C 180,E1 7194.019,E2 7194.019} C_VEL
LIN {X 0,Y 145.979,Z 1245.362,A -85,B 0,C 180,E1 7186.129,E2 7186.129} C_VEL
LIN {X 0,Y 150.59,Z 1251.255,A -85,B 0,C 180,E1 7175.69,E2 7175.69} C_VEL
LIN {X 0,Y 161.058,Z 1256.222,A -85,B 0,C 180,E1 7164.734,E2 7164.734} C_VEL
LIN {X 0,Y 175.764,Z 1259.449,A -85,B 0,C 180,E1 7155.796,E2 7155.796} C_VEL
LIN {X 0,Y 160.182,Z 1260.49,A -85,B 0,C 180,E1 7146.822,E2 7146.822} C_VEL
LIN {X 0,Y 150.005,Z 1259.971,A -85,B 0,C 180,E1 7136.105,E2 7136.105} C_VEL
LIN {X 0,Y 147.887,Z 1259.372,A -85,B 0,C 180,E1 7132.1,E2 7132.1} C_VEL
LIN {X 0,Y 145.856,Z 1258.554,A -85,B 0,C 180,E1 7129.196,E2 7129.196} C_VEL
LIN {X 0,Y 138.549,Z 1254.505,A -85,B 0,C 180,E1 7121.048,E2 7121.048} C_VEL
LIN {X 0,Y 138.038,Z 1253.292,A -85,B 0,C 180,E1 7118.563,E2 7118.563} C_VEL
LIN {X 0,Y 138.824,Z 1249.896,A -85,B 0,C 180,E1 7112.069,E2 7112.069} C_VEL
LIN {X 0,Y 138.928,Z 1246.628,A -85,B 0,C 180,E1 7107.531,E2 7107.531} C_VEL
LIN {X 0,Y 138.548,Z 1240.904,A -85,B 0,C 180,E1 7101.289,E2 7101.289} C_VEL
LIN {X 0,Y 138.608,Z 1235.684,A -85,B 0,C 180,E1 7096.234,E2 7096.234} C_VEL
LIN {X 0,Y 139.525,Z 1230.616,A -85,B 0,C 180,E1 7089.009,E2 7089.009} C_VEL
LIN {X 0,Y 142.085,Z 1223.986,A -85,B 0,C 180,E1 7082.331,E2 7082.331} C_VEL
LIN {X 0,Y 146.322,Z 1215.377,A -85,B 0,C 180,E1 7075.927,E2 7075.927} C_VEL
LIN {X 0,Y 151.743,Z 1205.268,A -85,B 0,C 180,E1 7070.278,E2 7070.278} C_VEL
LIN {X 0,Y 157.979,Z 1193.639,A -85,B 0,C 180,E1 7065.376,E2 7065.376} C_VEL
LIN {X 0,Y 164.372,Z 1180.883,A -85,B 0,C 180,E1 7061.308,E2 7061.308} C_VEL
LIN {X 0,Y 170.879,Z 1166.58,A -85,B 0,C 180,E1 7057.828,E2 7057.828} C_VEL
LIN {X 0,Y 176.673,Z 1152.084,A -85,B 0,C 180,E1 7055.143,E2 7055.143} C_VEL
LIN {X 0,Y 181.732,Z 1137.05,A -85,B 0,C 180,E1 7053.004,E2 7053.004} C_VEL
LIN {X 0,Y 184.971,Z 1126.395,A -85,B 0,C 180,E1 7051.764,E2 7051.764} C_VEL
LIN {X 0,Y 197.893,Z 1100.687,A -85,B 0,C 180,E1 7047.543,E2 7047.543} C_VEL
LIN {X 0,Y 213.402,Z 1068.829,A -85,B 0,C 180,E1 7043.566,E2 7043.566} C_VEL
LIN {X 0,Y 228.484,Z 1036.743,A -85,B 0,C 180,E1 7040.539,E2 7040.539} C_VEL
LIN {X 0,Y 236.507,Z 1018.479,A -85,B 0,C 180,E1 7039.126,E2 7039.126} C_VEL
LIN {X 0,Y 238.035,Z 990.426,A -85,B 0,C 180,E1 7034.969,E2 7034.969} C_VEL
LIN {X 0,Y 241.045,Z 961.174,A -85,B 0,C 180,E1 7031.243,E2 7031.243} C_VEL
LIN {X 0,Y 244.662,Z 934.145,A -85,B 0,C 180,E1 7028.342,E2 7028.342} C_VEL
LIN {X 0,Y 250.108,Z 897.462,A -85,B 0,C 180,E1 7025.117,E2 7025.117} C_VEL
LIN {X 0,Y 251.211,Z 889.063,A -85,B 0,C 180,E1 7024.394,E2 7024.394} C_VEL
LIN {X 0,Y 245.112,Z 874.265,A -85,B 0,C 180,E1 7020.195,E2 7020.195} C_VEL
LIN {X 0,Y 238.246,Z 858.443,A -85,B 0,C 180,E1 7014.944,E2 7014.944} C_VEL
LIN {X 0,Y 232.692,Z 845.752,A -85,B 0,C 180,E1 7010.034,E2 7010.034} C_VEL
LIN {X 0,Y 227.102,Z 832.865,A -85,B 0,C 180,E1 7004.158,E2 7004.158} C_VEL
LIN {X 0,Y 225.035,Z 827.96,A -85,B 0,C 180,E1 7001.476,E2 7001.476} C_VEL
LIN {X 0,Y 231.821,Z 826.332,A -85,B 0,C 180,E1 6997.158,E2 6997.158} C_VEL
LIN {X 0,Y 235.663,Z 826.075,A -85,B 0,C 180,E1 6994.928,E2 6994.928} C_VEL
LIN {X 0,Y 223.373,Z 875.313,A -85,B 0,C 180,E1 6990.008,E2 6990.008} C_VEL
LIN {X 0,Y 219.445,Z 892.849,A -85,B 0,C 180,E1 6988.27,E2 6988.27} C_VEL
LIN {X 0,Y 219.231,Z 899.01,A -85,B 0,C 180,E1 6987.976,E2 6987.976} C_VEL
LIN {X 0,Y 207.115,Z 1039.853,A -85,B 0,C 180,E1 6984.428,E2 6984.428} C_VEL
LIN {X 0,Y 204.997,Z 1067.458,A -85,B 0,C 180,E1 6983.437,E2 6983.437} C_VEL
LIN {X 0,Y 202.323,Z 1085.033,A -85,B 0,C 180,E1 6982.405,E2 6982.405} C_VEL
LIN {X 0,Y 198.595,Z 1101.3,A -85,B 0,C 180,E1 6981.06,E2 6981.06} C_VEL
LIN {X 0,Y 193.795,Z 1116.979,A -85,B 0,C 180,E1 6979.321,E2 6979.321} C_VEL
LIN {X 0,Y 188.126,Z 1131.633,A -85,B 0,C 180,E1 6977.171,E2 6977.171} C_VEL
LIN {X 0,Y 181.429,Z 1145.985,A -85,B 0,C 180,E1 6974.414,E2 6974.414} C_VEL
LIN {X 0,Y 174.501,Z 1158.692,A -85,B 0,C 180,E1 6971.213,E2 6971.213} C_VEL
LIN {X 0,Y 167.515,Z 1169.919,A -85,B 0,C 180,E1 6967.499,E2 6967.499} C_VEL
LIN {X 0,Y 160.692,Z 1179.701,A -85,B 0,C 180,E1 6963.194,E2 6963.194} C_VEL
LIN {X 0,Y 153.92,Z 1188.617,A -85,B 0,C 180,E1 6957.88,E2 6957.88} C_VEL
LIN {X 0,Y 148.374,Z 1195.518,A -85,B 0,C 180,E1 6952.166,E2 6952.166} C_VEL
LIN {X 0,Y 143.94,Z 1200.86,A -85,B 0,C 180,E1 6945.713,E2 6945.713} C_VEL
LIN {X 0,Y 140.934,Z 1204.535,A -85,B 0,C 180,E1 6938.563,E2 6938.563} C_VEL
LIN {X 0,Y 139.654,Z 1206.379,A -85,B 0,C 180,E1 6931.225,E2 6931.225} C_VEL
LIN {X 0,Y 139.945,Z 1206.458,A -85,B 0,C 180,E1 6924.254,E2 6924.254} C_VEL
LIN {X 0,Y 141.883,Z 1204.735,A -85,B 0,C 180,E1 6916.962,E2 6916.962} C_VEL
LIN {X 0,Y 145.583,Z 1201.163,A -85,B 0,C 180,E1 6909.91,E2 6909.91} C_VEL
LIN {X 0,Y 150.684,Z 1195.945,A -85,B 0,C 180,E1 6903.598,E2 6903.598} C_VEL
LIN {X 0,Y 157.082,Z 1188.847,A -85,B 0,C 180,E1 6897.844,E2 6897.844} C_VEL
LIN {X 0,Y 164.161,Z 1180.312,A -85,B 0,C 180,E1 6892.91,E2 6892.91} C_VEL
LIN {X 0,Y 171.987,Z 1169.849,A -85,B 0,C 180,E1 6888.483,E2 6888.483} C_VEL
LIN {X 0,Y 175.07,Z 1165.18,A -85,B 0,C 180,E1 6886.856,E2 6886.856} C_VEL
LIN {X 0,Y 170.171,Z 1165.974,A -85,B 0,C 180,E1 6885.315,E2 6885.315} C_VEL
LIN {X 0,Y 168.256,Z 1166.046,A -85,B 0,C 180,E1 6884.526,E2 6884.526} C_VEL
LIN {X 0,Y 163.92,Z 1166.934,A -85,B 0,C 180,E1 6883.093,E2 6883.093} C_VEL
LIN {X 0,Y 161.79,Z 1166.678,A -85,B 0,C 180,E1 6881.871,E2 6881.871} C_VEL
LIN {X 0,Y 153.242,Z 1183.099,A -85,B 0,C 180,E1 6875.501,E2 6875.501} C_VEL
LIN {X 0,Y 146.413,Z 1197.253,A -85,B 0,C 180,E1 6868.558,E2 6868.558} C_VEL
LIN {X 0,Y 141.215,Z 1209.994,A -85,B 0,C 180,E1 6860.734,E2 6860.734} C_VEL
LIN {X 0,Y 138.098,Z 1220.743,A -85,B 0,C 180,E1 6852.545,E2 6852.545} C_VEL
LIN {X 0,Y 136.796,Z 1229.812,A -85,B 0,C 180,E1 6844.192,E2 6844.192} C_VEL
LIN {X 0,Y 136.712,Z 1236.21,A -85,B 0,C 180,E1 6837.065,E2 6837.065} C_VEL
LIN {X 0,Y 137.349,Z 1241.894,A -85,B 0,C 180,E1 6829.514,E2 6829.514} C_VEL
LIN {X 0,Y 140.47,Z 1248.282,A -85,B 0,C 180,E1 6819.151,E2 6819.151} C_VEL
LIN {X 0,Y 149.067,Z 1254.17,A -85,B 0,C 180,E1 6807.547,E2 6807.547} C_VEL
LIN {X 0,Y 165.194,Z 1258.852,A -85,B 0,C 180,E1 6796.368,E2 6796.368} C_VEL
LIN {X 0,Y 165.954,Z 1259.035,A -85,B 0,C 180,E1 6795.812,E2 6795.812} C_VEL
LIN {X 0,Y 150.277,Z 1259.349,A -85,B 0,C 180,E1 6785.846,E2 6785.846} C_VEL
LIN {X 0,Y 140.959,Z 1258.01,A -85,B 0,C 180,E1 6774.3,E2 6774.3} C_VEL
LIN {X 0,Y 137.973,Z 1255.007,A -85,B 0,C 180,E1 6762.988,E2 6762.988} C_VEL
LIN {X 0,Y 138.038,Z 1253.292,A -85,B 0,C 180,E1 6758.563,E2 6758.563} C_VEL
LIN {X 0,Y 137.443,Z 1251.675,A -85,B 0,C 180,E1 6755.66,E2 6755.66} C_VEL
LIN {X 0,Y 135.097,Z 1248.805,A -85,B 0,C 180,E1 6751.977,E2 6751.977} C_VEL
LIN {X 0,Y 131.055,Z 1242.647,A -85,B 0,C 180,E1 6745.282,E2 6745.282} C_VEL
LIN {X 0,Y 130.915,Z 1241.785,A -85,B 0,C 180,E1 6744.351,E2 6744.351} C_VEL
LIN {X 0,Y 130.689,Z 1236.14,A -85,B 0,C 180,E1 6738.329,E2 6738.329} C_VEL
LIN {X 0,Y 131.088,Z 1231.928,A -85,B 0,C 180,E1 6730.86,E2 6730.86} C_VEL
LIN {X 0,Y 133.453,Z 1225.643,A -85,B 0,C 180,E1 6723.292,E2 6723.292} C_VEL
LIN {X 0,Y 137.527,Z 1217.811,A -85,B 0,C 180,E1 6716.465,E2 6716.465} C_VEL
LIN {X 0,Y 143.142,Z 1208.12,A -85,B 0,C 180,E1 6710.209,E2 6710.209} C_VEL
LIN {X 0,Y 149.66,Z 1196.998,A -85,B 0,C 180,E1 6704.92,E2 6704.92} C_VEL
LIN {X 0,Y 156.715,Z 1184.148,A -85,B 0,C 180,E1 6700.328,E2 6700.328} C_VEL
LIN {X 0,Y 163.742,Z 1170.207,A -85,B 0,C 180,E1 6696.591,E2 6696.591} C_VEL
LIN {X 0,Y 170.015,Z 1156.016,A -85,B 0,C 180,E1 6693.722,E2 6693.722} C_VEL
LIN {X 0,Y 175.729,Z 1140.873,A -85,B 0,C 180,E1 6691.416,E2 6691.416} C_VEL
LIN {X 0,Y 180.838,Z 1123.949,A -85,B 0,C 180,E1 6689.453,E2 6689.453} C_VEL
LIN {X 0,Y 182.864,Z 1116.657,A -85,B 0,C 180,E1 6688.818,E2 6688.818} C_VEL
LIN {X 0,Y 196.541,Z 1089.675,A -85,B 0,C 180,E1 6684.766,E2 6684.766} C_VEL
LIN {X 0,Y 212.235,Z 1057.889,A -85,B 0,C 180,E1 6681.133,E2 6681.133} C_VEL
LIN {X 0,Y 227.087,Z 1026.338,A -85,B 0,C 180,E1 6678.415,E2 6678.415} C_VEL
LIN {X 0,Y 230.149,Z 1019.239,A -85,B 0,C 180,E1 6677.849,E2 6677.849} C_VEL
LIN {X 0,Y 232.137,Z 990.924,A -85,B 0,C 180,E1 6673.577,E2 6673.577} C_VEL
LIN {X 0,Y 235.471,Z 962.716,A -85,B 0,C 180,E1 6669.91,E2 6669.91} C_VEL
LIN {X 0,Y 239.81,Z 933.091,A -85,B 0,C 180,E1 6666.704,E2 6666.704} C_VEL
LIN {X 0,Y 245.645,Z 896.894,A -85,B 0,C 180,E1 6663.5,E2 6663.5} C_VEL
LIN {X 0,Y 246.095,Z 893.078,A -85,B 0,C 180,E1 6663.144,E2 6663.144} C_VEL
LIN {X 0,Y 239.687,Z 877.203,A -85,B 0,C 180,E1 6658.446,E2 6658.446} C_VEL
LIN {X 0,Y 233.904,Z 863.541,A -85,B 0,C 180,E1 6653.742,E2 6653.742} C_VEL
LIN {X 0,Y 228.972,Z 851.972,A -85,B 0,C 180,E1 6649.177,E2 6649.177} C_VEL
LIN {X 0,Y 223.641,Z 839.407,A -85,B 0,C 180,E1 6643.373,E2 6643.373} C_VEL
LIN {X 0,Y 222.121,Z 835.683,A -85,B 0,C 180,E1 6641.36,E2 6641.36} C_VEL
LIN {X 0,Y 226.07,Z 834.361,A -85,B 0,C 180,E1 6638.735,E2 6638.735} C_VEL
LIN {X 0,Y 230.487,Z 833.614,A -85,B 0,C 180,E1 6636.049,E2 6636.049} C_VEL
LIN {X 0,Y 217.652,Z 883.839,A -85,B 0,C 180,E1 6631.054,E2 6631.054} C_VEL
LIN {X 0,Y 215.416,Z 893.798,A -85,B 0,C 180,E1 6630.083,E2 6630.083} C_VEL
LIN {X 0,Y 215.164,Z 899.983,A -85,B 0,C 180,E1 6629.785,E2 6629.785} C_VEL
LIN {X 0,Y 202.688,Z 1040.2,A -85,B 0,C 180,E1 6626.289,E2 6626.289} C_VEL
LIN {X 0,Y 200.414,Z 1068.428,A -85,B 0,C 180,E1 6625.273,E2 6625.273} C_VEL
LIN {X 0,Y 197.626,Z 1086,A -85,B 0,C 180,E1 6624.242,E2 6624.242} C_VEL
LIN {X 0,Y 193.709,Z 1102.422,A -85,B 0,C 180,E1 6622.884,E2 6622.884} C_VEL
LIN {X 0,Y 188.721,Z 1118.057,A -85,B 0,C 180,E1 6621.147,E2 6621.147} C_VEL
LIN {X 0,Y 182.535,Z 1133.326,A -85,B 0,C 180,E1 6618.885,E2 6618.885} C_VEL
LIN {X 0,Y 175.542,Z 1147.61,A -85,B 0,C 180,E1 6616.092,E2 6616.092} C_VEL
LIN {X 0,Y 168.032,Z 1160.681,A -85,B 0,C 180,E1 6612.709,E2 6612.709} C_VEL
LIN {X 0,Y 160.75,Z 1171.672,A -85,B 0,C 180,E1 6608.913,E2 6608.913} C_VEL
LIN {X 0,Y 153.15,Z 1181.928,A -85,B 0,C 180,E1 6604.151,E2 6604.151} C_VEL
LIN {X 0,Y 146.142,Z 1190.603,A -85,B 0,C 180,E1 6598.609,E2 6598.609} C_VEL
LIN {X 0,Y 140.407,Z 1197.224,A -85,B 0,C 180,E1 6592.61,E2 6592.61} C_VEL
LIN {X 0,Y 135.858,Z 1202.32,A -85,B 0,C 180,E1 6585.796,E2 6585.796} C_VEL
LIN {X 0,Y 132.844,Z 1205.807,A -85,B 0,C 180,E1 6578.216,E2 6578.216} C_VEL
LIN {X 0,Y 131.689,Z 1207.399,A -85,B 0,C 180,E1 6570.864,E2 6570.864} C_VEL
LIN {X 0,Y 132.105,Z 1207.343,A -85,B 0,C 180,E1 6563.475,E2 6563.475} C_VEL
LIN {X 0,Y 134.317,Z 1205.526,A -85,B 0,C 180,E1 6555.773,E2 6555.773} C_VEL
LIN {X 0,Y 138.134,Z 1202.098,A -85,B 0,C 180,E1 6548.776,E2 6548.776} C_VEL
LIN {X 0,Y 143.65,Z 1196.813,A -85,B 0,C 180,E1 6542.129,E2 6542.129} C_VEL
LIN {X 0,Y 150.527,Z 1189.621,A -85,B 0,C 180,E1 6536.133,E2 6536.133} C_VEL
LIN {X 0,Y 157.883,Z 1181.216,A -85,B 0,C 180,E1 6531.167,E2 6531.167} C_VEL
LIN {X 0,Y 165.736,Z 1171.111,A -85,B 0,C 180,E1 6526.76,E2 6526.76} C_VEL
LIN {X 0,Y 163.054,Z 1171.499,A -85,B 0,C 180,E1 6525.847,E2 6525.847} C_VEL
LIN {X 0,Y 158.251,Z 1172.123,A -85,B 0,C 180,E1 6524.029,E2 6524.029} C_VEL
LIN {X 0,Y 156.641,Z 1172.231,A -85,B 0,C 180,E1 6523.3,E2 6523.3} C_VEL
LIN {X 0,Y 152.859,Z 1172.952,A -85,B 0,C 180,E1 6521.852,E2 6521.852} C_VEL
LIN {X 0,Y 150.701,Z 1172.935,A -85,B 0,C 180,E1 6520.434,E2 6520.434} C_VEL
LIN {X 0,Y 142.143,Z 1189.235,A -85,B 0,C 180,E1 6513.157,E2 6513.157} C_VEL
LIN {X 0,Y 135.741,Z 1202.974,A -85,B 0,C 180,E1 6505.293,E2 6505.293} C_VEL
LIN {X 0,Y 131.435,Z 1214.85,A -85,B 0,C 180,E1 6496.803,E2 6496.803} C_VEL
LIN {X 0,Y 129.241,Z 1224.973,A -85,B 0,C 180,E1 6487.954,E2 6487.954} C_VEL
LIN {X 0,Y 128.766,Z 1232.464,A -85,B 0,C 180,E1 6480,E2 6480} C_VEL
LIN {X 0,Y 129.07,Z 1238.466,A -85,B 0,C 180,E1 6472.432,E2 6472.432} C_VEL
LIN {X 0,Y 130.999,Z 1244.877,A -85,B 0,C 180,E1 6462.682,E2 6462.682} C_VEL
LIN {X 0,Y 137.534,Z 1251.315,A -85,B 0,C 180,E1 6450.85,E2 6450.85} C_VEL
LIN {X 0,Y 151.081,Z 1256.831,A -85,B 0,C 180,E1 6439.065,E2 6439.065} C_VEL
LIN {X 0,Y 156.346,Z 1258.214,A -85,B 0,C 180,E1 6435.886,E2 6435.886} C_VEL
LIN {X 0,Y 140.876,Z 1257.821,A -85,B 0,C 180,E1 6425.1,E2 6425.1} C_VEL
LIN {X 0,Y 132.295,Z 1255.728,A -85,B 0,C 180,E1 6412.678,E2 6412.678} C_VEL
LIN {X 0,Y 130.219,Z 1252.325,A -85,B 0,C 180,E1 6401.522,E2 6401.522} C_VEL
LIN {X 0,Y 130.884,Z 1248.814,A -85,B 0,C 180,E1 6393.948,E2 6393.948} C_VEL
LIN {X 0,Y 131.239,Z 1246.055,A -85,B 0,C 180,E1 6389.569,E2 6389.569} C_VEL
LIN {X 0,Y 130.915,Z 1241.785,A -85,B 0,C 180,E1 6384.351,E2 6384.351} C_VEL
LIN {X 0,Y 129.982,Z 1239.454,A -85,B 0,C 180,E1 6381.652,E2 6381.652} C_VEL
LIN {X 0,Y 126.762,Z 1236.173,A -85,B 0,C 180,E1 6377.381,E2 6377.381} C_VEL
LIN {X 0,Y 123.437,Z 1232.457,A -85,B 0,C 180,E1 6371.89,E2 6371.89} C_VEL
LIN {X 0,Y 123.362,Z 1230.78,A -85,B 0,C 180,E1 6369.405,E2 6369.405} C_VEL
LIN {X 0,Y 126.083,Z 1224.616,A -85,B 0,C 180,E1 6361.595,E2 6361.595} C_VEL
LIN {X 0,Y 130.661,Z 1216.773,A -85,B 0,C 180,E1 6354.445,E2 6354.445} C_VEL
LIN {X 0,Y 136.559,Z 1207.497,A -85,B 0,C 180,E1 6348.226,E2 6348.226} C_VEL
LIN {X 0,Y 143.367,Z 1196.814,A -85,B 0,C 180,E1 6342.929,E2 6342.929} C_VEL
LIN {X 0,Y 150.874,Z 1184.124,A -85,B 0,C 180,E1 6338.258,E2 6338.258} C_VEL
LIN {X 0,Y 158.293,Z 1170.373,A -85,B 0,C 180,E1 6334.49,E2 6334.49} C_VEL
LIN {X 0,Y 165.281,Z 1155.631,A -85,B 0,C 180,E1 6331.471,E2 6331.471} C_VEL
LIN {X 0,Y 171.284,Z 1140.664,A -85,B 0,C 180,E1 6329.199,E2 6329.199} C_VEL
LIN {X 0,Y 176.405,Z 1124.703,A -85,B 0,C 180,E1 6327.331,E2 6327.331} C_VEL
LIN {X 0,Y 180.605,Z 1108.149,A -85,B 0,C 180,E1 6325.99,E2 6325.99} C_VEL
LIN {X 0,Y 181.869,Z 1105.228,A -85,B 0,C 180,E1 6325.636,E2 6325.636} C_VEL
LIN {X 0,Y 198.137,Z 1073.418,A -85,B 0,C 180,E1 6321.411,E2 6321.411} C_VEL
LIN {X 0,Y 214.177,Z 1040.921,A -85,B 0,C 180,E1 6318.202,E2 6318.202} C_VEL
LIN {X 0,Y 223.812,Z 1020.504,A -85,B 0,C 180,E1 6316.614,E2 6316.614} C_VEL
LIN {X 0,Y 226.244,Z 992.276,A -85,B 0,C 180,E1 6312.248,E2 6312.248} C_VEL
LIN {X 0,Y 229.957,Z 963.913,A -85,B 0,C 180,E1 6308.502,E2 6308.502} C_VEL
LIN {X 0,Y 234.71,Z 934.312,A -85,B 0,C 180,E1 6305.243,E2 6305.243} C_VEL
LIN {X 0,Y 240.935,Z 898.462,A -85,B 0,C 180,E1 6302.023,E2 6302.023} C_VEL
LIN {X 0,Y 241.081,Z 897.231,A -85,B 0,C 180,E1 6301.901,E2 6301.901} C_VEL
LIN {X 0,Y 235.181,Z 882.258,A -85,B 0,C 180,E1 6297.319,E2 6297.319} C_VEL
LIN {X 0,Y 230.052,Z 869.773,A -85,B 0,C 180,E1 6292.947,E2 6292.947} C_VEL
LIN {X 0,Y 225.455,Z 858.622,A -85,B 0,C 180,E1 6288.488,E2 6288.488} C_VEL
LIN {X 0,Y 220.217,Z 845.948,A -85,B 0,C 180,E1 6282.562,E2 6282.562} C_VEL
LIN {X 0,Y 219.282,Z 843.349,A -85,B 0,C 180,E1 6281.11,E2 6281.11} C_VEL
LIN {X 0,Y 222.58,Z 841.991,A -85,B 0,C 180,E1 6278.938,E2 6278.938} C_VEL
LIN {X 0,Y 225.268,Z 841.589,A -85,B 0,C 180,E1 6277.188,E2 6277.188} C_VEL
LIN {X 0,Y 212.115,Z 891.723,A -85,B 0,C 180,E1 6272.227,E2 6272.227} C_VEL
LIN {X 0,Y 211.599,Z 895.452,A -85,B 0,C 180,E1 6271.917,E2 6271.917} C_VEL
LIN {X 0,Y 211.282,Z 901.336,A -85,B 0,C 180,E1 6271.653,E2 6271.653} C_VEL
LIN {X 0,Y 198.483,Z 1040.548,A -85,B 0,C 180,E1 6268.231,E2 6268.231} C_VEL
LIN {X 0,Y 196.067,Z 1069.245,A -85,B 0,C 180,E1 6267.201,E2 6267.201} C_VEL
LIN {X 0,Y 193.185,Z 1086.761,A -85,B 0,C 180,E1 6266.181,E2 6266.181} C_VEL
LIN {X 0,Y 189.162,Z 1103.071,A -85,B 0,C 180,E1 6264.845,E2 6264.845} C_VEL
LIN {X 0,Y 183.85,Z 1119.133,A -85,B 0,C 180,E1 6263.072,E2 6263.072} C_VEL
LIN {X 0,Y 177.386,Z 1134.449,A -85,B 0,C 180,E1 6260.802,E2 6260.802} C_VEL
LIN {X 0,Y 170.137,Z 1148.647,A -85,B 0,C 180,E1 6258.017,E2 6258.017} C_VEL
LIN {X 0,Y 162.899,Z 1160.739,A -85,B 0,C 180,E1 6254.893,E2 6254.893} C_VEL
LIN {X 0,Y 155.222,Z 1171.933,A -85,B 0,C 180,E1 6251.068,E2 6251.068} C_VEL
LIN {X 0,Y 147.661,Z 1181.697,A -85,B 0,C 180,E1 6246.569,E2 6246.569} C_VEL
LIN {X 0,Y 140.078,Z 1190.597,A -85,B 0,C 180,E1 6240.92,E2 6240.92} C_VEL
LIN {X 0,Y 133.798,Z 1197.483,A -85,B 0,C 180,E1 6234.733,E2 6234.733} C_VEL
LIN {X 0,Y 128.719,Z 1202.804,A -85,B 0,C 180,E1 6227.628,E2 6227.628} C_VEL
LIN {X 0,Y 125.249,Z 1206.464,A -85,B 0,C 180,E1 6219.645,E2 6219.645} C_VEL
LIN {X 0,Y 123.772,Z 1208.295,A -85,B 0,C 180,E1 6211.382,E2 6211.382} C_VEL
LIN {X 0,Y 124.138,Z 1208.355,A -85,B 0,C 180,E1 6203.519,E2 6203.519} C_VEL
LIN {X 0,Y 126.434,Z 1206.619,A -85,B 0,C 180,E1 6195.335,E2 6195.335} C_VEL
LIN {X 0,Y 130.745,Z 1203.033,A -85,B 0,C 180,E1 6187.513,E2 6187.513} C_VEL
LIN {X 0,Y 136.603,Z 1197.794,A -85,B 0,C 180,E1 6180.626,E2 6180.626} C_VEL
LIN {X 0,Y 143.564,Z 1190.973,A -85,B 0,C 180,E1 6174.679,E2 6174.679} C_VEL
LIN {X 0,Y 151.911,Z 1181.954,A -85,B 0,C 180,E1 6169.196,E2 6169.196} C_VEL
LIN {X 0,Y 156.253,Z 1176.767,A -85,B 0,C 180,E1 6166.725,E2 6166.725} C_VEL
LIN {X 0,Y 151.664,Z 1177.258,A -85,B 0,C 180,E1 6164.864,E2 6164.864} C_VEL
LIN {X 0,Y 146.978,Z 1177.877,A -85,B 0,C 180,E1 6162.868,E2 6162.868} C_VEL
LIN {X 0,Y 145.104,Z 1178.013,A -85,B 0,C 180,E1 6161.902,E2 6161.902} C_VEL
LIN {X 0,Y 141.299,Z 1178.599,A -85,B 0,C 180,E1 6160.088,E2 6160.088} C_VEL
LIN {X 0,Y 139.681,Z 1178.65,A -85,B 0,C 180,E1 6158.782,E2 6158.782} C_VEL
LIN {X 0,Y 131.413,Z 1194.482,A -85,B 0,C 180,E1 6150.65,E2 6150.65} C_VEL
LIN {X 0,Y 125.634,Z 1207.654,A -85,B 0,C 180,E1 6141.967,E2 6141.967} C_VEL
LIN {X 0,Y 122.213,Z 1218.88,A -85,B 0,C 180,E1 6132.762,E2 6132.762} C_VEL
LIN {X 0,Y 120.946,Z 1227.782,A -85,B 0,C 180,E1 6123.792,E2 6123.792} C_VEL
LIN {X 0,Y 120.935,Z 1234.158,A -85,B 0,C 180,E1 6116.207,E2 6116.207} C_VEL
LIN {X 0,Y 121.799,Z 1240.198,A -85,B 0,C 180,E1 6107.676,E2 6107.676} C_VEL
LIN {X 0,Y 126.038,Z 1247.247,A -85,B 0,C 180,E1 6095.636,E2 6095.636} C_VEL
LIN {X 0,Y 137.015,Z 1253.833,A -85,B 0,C 180,E1 6082.706,E2 6082.706} C_VEL
LIN {X 0,Y 146.669,Z 1257.032,A -85,B 0,C 180,E1 6075.871,E2 6075.871} C_VEL
LIN {X 0,Y 131.575,Z 1255.93,A -85,B 0,C 180,E1 6064.225,E2 6064.225} C_VEL
LIN {X 0,Y 123.96,Z 1253.216,A -85,B 0,C 180,E1 6051.29,E2 6051.29} C_VEL
LIN {X 0,Y 122.567,Z 1249.556,A -85,B 0,C 180,E1 6040.345,E2 6040.345} C_VEL
LIN {X 0,Y 123.357,Z 1245.896,A -85,B 0,C 180,E1 6032.794,E2 6032.794} C_VEL
LIN {X 0,Y 123.455,Z 1242.787,A -85,B 0,C 180,E1 6028.15,E2 6028.15} C_VEL
LIN {X 0,Y 122.96,Z 1236.687,A -85,B 0,C 180,E1 6021.118,E2 6021.118} C_VEL
LIN {X 0,Y 122.924,Z 1232.352,A -85,B 0,C 180,E1 6012.002,E2 6012.002} C_VEL
LIN {X 0,Y 123.362,Z 1230.78,A -85,B 0,C 180,E1 6009.405,E2 6009.405} C_VEL
LIN {X 0,Y 123.329,Z 1228.38,A -85,B 0,C 180,E1 6005.978,E2 6005.978} C_VEL
LIN {X 0,Y 121.364,Z 1221.231,A -85,B 0,C 180,E1 5997.179,E2 5997.179} C_VEL
LIN {X 0,Y 122.574,Z 1217.828,A -85,B 0,C 180,E1 5993.939,E2 5993.939} C_VEL
LIN {X 0,Y 129.038,Z 1208.452,A -85,B 0,C 180,E1 5987.017,E2 5987.017} C_VEL
LIN {X 0,Y 136.71,Z 1197.399,A -85,B 0,C 180,E1 5981.129,E2 5981.129} C_VEL
LIN {X 0,Y 144.62,Z 1185.144,A -85,B 0,C 180,E1 5976.355,E2 5976.355} C_VEL
LIN {X 0,Y 152.348,Z 1171.866,A -85,B 0,C 180,E1 5972.56,E2 5972.56} C_VEL
LIN {X 0,Y 160.043,Z 1156.794,A -85,B 0,C 180,E1 5969.373,E2 5969.373} C_VEL
LIN {X 0,Y 166.255,Z 1142.508,A -85,B 0,C 180,E1 5967.126,E2 5967.126} C_VEL
LIN {X 0,Y 171.864,Z 1126.716,A -85,B 0,C 180,E1 5965.231,E2 5965.231} C_VEL
LIN {X 0,Y 176.613,Z 1109.389,A -85,B 0,C 180,E1 5963.777,E2 5963.777} C_VEL
LIN {X 0,Y 179.273,Z 1097.34,A -85,B 0,C 180,E1 5963.046,E2 5963.046} C_VEL
LIN {X 0,Y 196.162,Z 1064.791,A -85,B 0,C 180,E1 5959.011,E2 5959.011} C_VEL
LIN {X 0,Y 212.897,Z 1031.096,A -85,B 0,C 180,E1 5955.948,E2 5955.948} C_VEL
LIN {X 0,Y 217.605,Z 1020.955,A -85,B 0,C 180,E1 5955.184,E2 5955.184} C_VEL
LIN {X 0,Y 220.683,Z 991.339,A -85,B 0,C 180,E1 5950.541,E2 5950.541} C_VEL
LIN {X 0,Y 224.88,Z 962.855,A -85,B 0,C 180,E1 5946.767,E2 5946.767} C_VEL
LIN {X 0,Y 230.164,Z 933.059,A -85,B 0,C 180,E1 5943.487,E2 5943.487} C_VEL
LIN {X 0,Y 236.065,Z 901.23,A -85,B 0,C 180,E1 5940.59,E2 5940.59} C_VEL
LIN {X 0,Y 230.754,Z 887.565,A -85,B 0,C 180,E1 5936.273,E2 5936.273} C_VEL
LIN {X 0,Y 226.137,Z 875.771,A -85,B 0,C 180,E1 5932.04,E2 5932.04} C_VEL
LIN {X 0,Y 221.622,Z 864.596,A -85,B 0,C 180,E1 5927.493,E2 5927.493} C_VEL
LIN {X 0,Y 216.827,Z 852.49,A -85,B 0,C 180,E1 5921.725,E2 5921.725} C_VEL
LIN {X 0,Y 216.346,Z 851.182,A -85,B 0,C 180,E1 5920.984,E2 5920.984} C_VEL
LIN {X 0,Y 219.57,Z 849.617,A -85,B 0,C 180,E1 5918.915,E2 5918.915} C_VEL
LIN {X 0,Y 220.313,Z 849.41,A -85,B 0,C 180,E1 5918.431,E2 5918.431} C_VEL
LIN {X 0,Y 208.049,Z 895.415,A -85,B 0,C 180,E1 5913.927,E2 5913.927} C_VEL
LIN {X 0,Y 207.732,Z 901.676,A -85,B 0,C 180,E1 5913.612,E2 5913.612} C_VEL
LIN {X 0,Y 194.517,Z 1040.896,A -85,B 0,C 180,E1 5910.255,E2 5910.255} C_VEL
LIN {X 0,Y 191.931,Z 1070.215,A -85,B 0,C 180,E1 5909.206,E2 5909.206} C_VEL
LIN {X 0,Y 188.928,Z 1087.745,A -85,B 0,C 180,E1 5908.193,E2 5908.193} C_VEL
LIN {X 0,Y 184.575,Z 1104.663,A -85,B 0,C 180,E1 5906.813,E2 5906.813} C_VEL
LIN {X 0,Y 179.197,Z 1120.208,A -85,B 0,C 180,E1 5905.1,E2 5905.1} C_VEL
LIN {X 0,Y 172.483,Z 1135.501,A -85,B 0,C 180,E1 5902.845,E2 5902.845} C_VEL
LIN {X 0,Y 164.936,Z 1149.683,A -85,B 0,C 180,E1 5900.066,E2 5900.066} C_VEL
LIN {X 0,Y 157.378,Z 1161.762,A -85,B 0,C 180,E1 5896.932,E2 5896.932} C_VEL
LIN {X 0,Y 149.329,Z 1172.94,A -85,B 0,C 180,E1 5893.069,E2 5893.069} C_VEL
LIN {X 0,Y 141.364,Z 1182.695,A -85,B 0,C 180,E1 5888.487,E2 5888.487} C_VEL
LIN {X 0,Y 133.328,Z 1191.587,A -85,B 0,C 180,E1 5882.674,E2 5882.674} C_VEL
LIN {X 0,Y 126.627,Z 1198.466,A -85,B 0,C 180,E1 5876.237,E2 5876.237} C_VEL
LIN {X 0,Y 121.173,Z 1203.775,A -85,B 0,C 180,E1 5868.766,E2 5868.766} C_VEL
LIN {X 0,Y 117.426,Z 1207.429,A -85,B 0,C 180,E1 5860.294,E2 5860.294} C_VEL
LIN {X 0,Y 115.832,Z 1209.253,A -85,B 0,C 180,E1 5851.477,E2 5851.477} C_VEL
LIN {X 0,Y 116.243,Z 1209.303,A -85,B 0,C 180,E1 5843.077,E2 5843.077} C_VEL
LIN {X 0,Y 118.754,Z 1207.561,A -85,B 0,C 180,E1 5834.363,E2 5834.363} C_VEL
LIN {X 0,Y 123.426,Z 1203.968,A -85,B 0,C 180,E1 5826.099,E2 5826.099} C_VEL
LIN {X 0,Y 129.723,Z 1198.717,A -85,B 0,C 180,E1 5818.901,E2 5818.901} C_VEL
LIN {X 0,Y 137.144,Z 1191.887,A -85,B 0,C 180,E1 5812.755,E2 5812.755} C_VEL
LIN {X 0,Y 145.821,Z 1183.024,A -85,B 0,C 180,E1 5807.241,E2 5807.241} C_VEL
LIN {X 0,Y 146.849,Z 1181.891,A -85,B 0,C 180,E1 5806.624,E2 5806.624} C_VEL
LIN {X 0,Y 141.613,Z 1182.495,A -85,B 0,C 180,E1 5804.348,E2 5804.348} C_VEL
LIN {X 0,Y 135.77,Z 1183.239,A -85,B 0,C 180,E1 5801.515,E2 5801.515} C_VEL
LIN {X 0,Y 133.775,Z 1183.391,A -85,B 0,C 180,E1 5800.316,E2 5800.316} C_VEL
LIN {X 0,Y 130.36,Z 1183.917,A -85,B 0,C 180,E1 5798.411,E2 5798.411} C_VEL
LIN {X 0,Y 128.832,Z 1183.891,A -85,B 0,C 180,E1 5796.977,E2 5796.977} C_VEL
LIN {X 0,Y 121.098,Z 1198.944,A -85,B 0,C 180,E1 5788.076,E2 5788.076} C_VEL
LIN {X 0,Y 116.055,Z 1211.406,A -85,B 0,C 180,E1 5778.589,E2 5778.589} C_VEL
LIN {X 0,Y 113.502,Z 1221.992,A -85,B 0,C 180,E1 5768.613,E2 5768.613} C_VEL
LIN {X 0,Y 112.984,Z 1229.6,A -85,B 0,C 180,E1 5760,E2 5760} C_VEL
LIN {X 0,Y 113.352,Z 1235.663,A -85,B 0,C 180,E1 5751.886,E2 5751.886} C_VEL
LIN {X 0,Y 115.48,Z 1242.309,A -85,B 0,C 180,E1 5741.315,E2 5741.315} C_VEL
LIN {X 0,Y 122.93,Z 1249.427,A -85,B 0,C 180,E1 5728.082,E2 5728.082} C_VEL
LIN {X 0,Y 137.093,Z 1255.488,A -85,B 0,C 180,E1 5715.847,E2 5715.847} C_VEL
LIN {X 0,Y 122.385,Z 1253.68,A -85,B 0,C 180,E1 5703.195,E2 5703.195} C_VEL
LIN {X 0,Y 115.771,Z 1250.4,A -85,B 0,C 180,E1 5689.691,E2 5689.691} C_VEL
LIN {X 0,Y 115.067,Z 1246.315,A -85,B 0,C 180,E1 5678.502,E2 5678.502} C_VEL
LIN {X 0,Y 115.813,Z 1243.019,A -85,B 0,C 180,E1 5671.986,E2 5671.986} C_VEL
LIN {X 0,Y 115.626,Z 1239.561,A -85,B 0,C 180,E1 5667.033,E2 5667.033} C_VEL
LIN {X 0,Y 115.198,Z 1236.08,A -85,B 0,C 180,E1 5662.526,E2 5662.526} C_VEL
LIN {X 0,Y 114.749,Z 1232.9,A -85,B 0,C 180,E1 5653.816,E2 5653.816} C_VEL
LIN {X 0,Y 116.482,Z 1227.903,A -85,B 0,C 180,E1 5645.134,E2 5645.134} C_VEL
LIN {X 0,Y 120.449,Z 1221.057,A -85,B 0,C 180,E1 5636.976,E2 5636.976} C_VEL
LIN {X 0,Y 122.574,Z 1217.828,A -85,B 0,C 180,E1 5633.939,E2 5633.939} C_VEL
LIN {X 0,Y 124.116,Z 1214.267,A -85,B 0,C 180,E1 5630.817,E2 5630.817} C_VEL
LIN {X 0,Y 126.196,Z 1204.518,A -85,B 0,C 180,E1 5622.789,E2 5622.789} C_VEL
LIN {X 0,Y 128.676,Z 1200.056,A -85,B 0,C 180,E1 5620.161,E2 5620.161} C_VEL
LIN {X 0,Y 137.234,Z 1187.939,A -85,B 0,C 180,E1 5614.959,E2 5614.959} C_VEL
LIN {X 0,Y 145.981,Z 1174.302,A -85,B 0,C 180,E1 5610.74,E2 5610.74} C_VEL
LIN {X 0,Y 153.912,Z 1160.175,A -85,B 0,C 180,E1 5607.542,E2 5607.542} C_VEL
LIN {X 0,Y 161.105,Z 1145.03,A -85,B 0,C 180,E1 5605.035,E2 5605.035} C_VEL
LIN {X 0,Y 167.362,Z 1128.999,A -85,B 0,C 180,E1 5603.079,E2 5603.079} C_VEL
LIN {X 0,Y 172.532,Z 1111.956,A -85,B 0,C 180,E1 5601.555,E2 5601.555} C_VEL
LIN {X 0,Y 176.276,Z 1094.808,A -85,B 0,C 180,E1 5600.52,E2 5600.52} C_VEL
LIN {X 0,Y 177.473,Z 1088.232,A -85,B 0,C 180,E1 5600.285,E2 5600.285} C_VEL
LIN {X 0,Y 194.999,Z 1054.87,A -85,B 0,C 180,E1 5596.506,E2 5596.506} C_VEL
LIN {X 0,Y 211.432,Z 1021.667,A -85,B 0,C 180,E1 5593.747,E2 5593.747} C_VEL
LIN {X 0,Y 214.77,Z 993.866,A -85,B 0,C 180,E1 5589.279,E2 5589.279} C_VEL
LIN {X 0,Y 219.595,Z 963.858,A -85,B 0,C 180,E1 5585.225,E2 5585.225} C_VEL
LIN {X 0,Y 225.385,Z 933.442,A -85,B 0,C 180,E1 5581.849,E2 5581.849} C_VEL
LIN {X 0,Y 230.977,Z 905.291,A -85,B 0,C 180,E1 5579.254,E2 5579.254} C_VEL
LIN {X 0,Y 226.347,Z 892.827,A -85,B 0,C 180,E1 5575.185,E2 5575.185} C_VEL
LIN {X 0,Y 221.899,Z 881.198,A -85,B 0,C 180,E1 5570.926,E2 5570.926} C_VEL
LIN {X 0,Y 217.817,Z 870.546,A -85,B 0,C 180,E1 5566.46,E2 5566.46} C_VEL
LIN {X 0,Y 213.542,Z 859.322,A -85,B 0,C 180,E1 5561.044,E2 5561.044} C_VEL
LIN {X 0,Y 213.567,Z 858.875,A -85,B 0,C 180,E1 5560.727,E2 5560.727} C_VEL
LIN {X 0,Y 215.268,Z 857.873,A -85,B 0,C 180,E1 5559.648,E2 5559.648} C_VEL
LIN {X 0,Y 204.729,Z 896.363,A -85,B 0,C 180,E1 5555.939,E2 5555.939} C_VEL
LIN {X 0,Y 204.367,Z 902.672,A -85,B 0,C 180,E1 5555.622,E2 5555.622} C_VEL
LIN {X 0,Y 190.803,Z 1041.243,A -85,B 0,C 180,E1 5552.36,E2 5552.36} C_VEL
LIN {X 0,Y 188.062,Z 1071.032,A -85,B 0,C 180,E1 5551.305,E2 5551.305} C_VEL
LIN {X 0,Y 184.972,Z 1088.466,A -85,B 0,C 180,E1 5550.313,E2 5550.313} C_VEL
LIN {X 0,Y 180.724,Z 1104.558,A -85,B 0,C 180,E1 5549.033,E2 5549.033} C_VEL
LIN {X 0,Y 175.049,Z 1120.633,A -85,B 0,C 180,E1 5547.314,E2 5547.314} C_VEL
LIN {X 0,Y 168.176,Z 1135.841,A -85,B 0,C 180,E1 5545.123,E2 5545.123} C_VEL
LIN {X 0,Y 160.31,Z 1150.13,A -85,B 0,C 180,E1 5542.376,E2 5542.376} C_VEL
LIN {X 0,Y 152.07,Z 1162.786,A -85,B 0,C 180,E1 5539.117,E2 5539.117} C_VEL
LIN {X 0,Y 143.633,Z 1173.947,A -85,B 0,C 180,E1 5535.231,E2 5535.231} C_VEL
LIN {X 0,Y 135.239,Z 1183.693,A -85,B 0,C 180,E1 5530.581,E2 5530.581} C_VEL
LIN {X 0,Y 126.716,Z 1192.578,A -85,B 0,C 180,E1 5524.612,E2 5524.612} C_VEL
LIN {X 0,Y 119.555,Z 1199.449,A -85,B 0,C 180,E1 5517.92,E2 5517.92} C_VEL
LIN {X 0,Y 113.681,Z 1204.747,A -85,B 0,C 180,E1 5510.054,E2 5510.054} C_VEL
LIN {X 0,Y 109.621,Z 1208.394,A -85,B 0,C 180,E1 5501.036,E2 5501.036} C_VEL
LIN {X 0,Y 107.892,Z 1210.211,A -85,B 0,C 180,E1 5491.586,E2 5491.586} C_VEL
LIN {X 0,Y 108.357,Z 1210.252,A -85,B 0,C 180,E1 5482.57,E2 5482.57} C_VEL
LIN {X 0,Y 111.113,Z 1208.503,A -85,B 0,C 180,E1 5473.257,E2 5473.257} C_VEL
LIN {X 0,Y 116.193,Z 1204.903,A -85,B 0,C 180,E1 5464.508,E2 5464.508} C_VEL
LIN {X 0,Y 122.973,Z 1199.641,A -85,B 0,C 180,E1 5456.984,E2 5456.984} C_VEL
LIN {X 0,Y 130.894,Z 1192.801,A -85,B 0,C 180,E1 5450.645,E2 5450.645} C_VEL
LIN {X 0,Y 137.187,Z 1186.767,A -85,B 0,C 180,E1 5446.517,E2 5446.517} C_VEL
LIN {X 0,Y 130.186,Z 1187.585,A -85,B 0,C 180,E1 5443.123,E2 5443.123} C_VEL
LIN {X 0,Y 124.08,Z 1188.3,A -85,B 0,C 180,E1 5439.54,E2 5439.54} C_VEL
LIN {X 0,Y 122.397,Z 1188.477,A -85,B 0,C 180,E1 5438.38,E2 5438.38} C_VEL
LIN {X 0,Y 119.041,Z 1188.949,A -85,B 0,C 180,E1 5436.013,E2 5436.013} C_VEL
LIN {X 0,Y 117.865,Z 1189.071,A -85,B 0,C 180,E1 5434.615,E2 5434.615} C_VEL
LIN {X 0,Y 110.986,Z 1203.002,A -85,B 0,C 180,E1 5425.052,E2 5425.052} C_VEL
LIN {X 0,Y 106.788,Z 1214.916,A -85,B 0,C 180,E1 5414.644,E2 5414.644} C_VEL
